LIN {X 0,Y 377.253,Z 474.78,A -85,B 0,C 180,E1 17667.471,E2 17667.471} C_VEL
LIN {X 0,Y 377.352,Z 476.669,A -85,B 0,C 180,E1 17678.06,E2 17678.06} C_VEL
LIN {X 0,Y 405.351,Z 515.448,A -85,B 0,C 180,E1 17684.462,E2 17684.462} C_VEL
LIN {X 0,Y 431.336,Z 545.833,A -85,B 0,C 180,E1 17691.711,E2 17691.711} C_VEL
LIN {X 0,Y 454.819,Z 571.984,A -85,B 0,C 180,E1 17699.556,E2 17699.556} C_VEL
LIN {X 0,Y 473.643,Z 591.464,A -85,B 0,C 180,E1 17707.256,E2 17707.256} C_VEL
LIN {X 0,Y 486.809,Z 605.487,A -85,B 0,C 180,E1 17714.646,E2 17714.646} C_VEL
LIN {X 0,Y 493.723,Z 611.989,A -85,B 0,C 180,E1 17720.274,E2 17720.274} C_VEL
LIN {X 0,Y 498.301,Z 615.614,A -85,B 0,C 180,E1 17727.82,E2 17727.82} C_VEL
LIN {X 0,Y 497.056,Z 614.877,A -85,B 0,C 180,E1 17735.239,E2 17735.239} C_VEL
LIN {X 0,Y 492.043,Z 609.419,A -85,B 0,C 180,E1 17741.556,E2 17741.556} C_VEL
LIN {X 0,Y 481.093,Z 598.897,A -85,B 0,C 180,E1 17748.962,E2 17748.962} C_VEL
LIN {X 0,Y 464.615,Z 582.345,A -85,B 0,C 180,E1 17756.667,E2 17756.667} C_VEL
LIN {X 0,Y 442.794,Z 559.28,A -85,B 0,C 180,E1 17764.614,E2 17764.614} C_VEL
LIN {X 0,Y 416.817,Z 529.891,A -85,B 0,C 180,E1 17772.484,E2 17772.484} C_VEL
LIN {X 0,Y 391.726,Z 498.659,A -85,B 0,C 180,E1 17778.671,E2 17778.671} C_VEL
LIN {X 0,Y 376.899,Z 474.78,A -85,B 0,C 180,E1 17782.231,E2 17782.231} C_VEL
LIN {X 0,Y 377.23,Z 474.78,A -85,B 0,C 180,E1 17792.527,E2 17792.527} C_VEL
LIN {X 0,Y 377.899,Z 474.78,A -85,B 0,C 180,E1 17802.548,E2 17802.548} C_VEL
LIN {X 0,Y 378.35,Z 474.78,A -85,B 0,C 180,E1 17812.001,E2 17812.001} C_VEL
LIN {X 0,Y 378.531,Z 474.78,A -85,B 0,C 180,E1 17821.217,E2 17821.217} C_VEL
LIN {X 0,Y 378.086,Z 474.78,A -85,B 0,C 180,E1 17830.677,E2 17830.677} C_VEL
LIN {X 0,Y 377.317,Z 474.78,A -85,B 0,C 180,E1 17842.532,E2 17842.532} C_VEL
LIN {X 0,Y 376.834,Z 474.78,A -85,B 0,C 180,E1 17853.007,E2 17853.007} C_VEL
LIN {X 0,Y 376.964,Z 476.24,A -85,B 0,C 180,E1 17857.663,E2 17857.663} C_VEL
LIN {X 0,Y 410.937,Z 533.681,A -85,B 0,C 180,E1 17865.009,E2 17865.009} C_VEL
LIN {X 0,Y 427.352,Z 580.89,A -85,B 0,C 180,E1 17869.565,E2 17869.565} C_VEL
LIN {X 0,Y 414.888,Z 639.247,A -85,B 0,C 180,E1 17873.387,E2 17873.387} C_VEL
LIN {X 0,Y 400.436,Z 690.553,A -85,B 0,C 180,E1 17879.252,E2 17879.252} C_VEL
LIN {X 0,Y 388.051,Z 731.295,A -85,B 0,C 180,E1 17887.04,E2 17887.04} C_VEL
LIN {X 0,Y 381.14,Z 758.804,A -85,B 0,C 180,E1 17896.188,E2 17896.188} C_VEL
LIN {X 0,Y 379.523,Z 770.88,A -85,B 0,C 180,E1 17904.267,E2 17904.267} C_VEL
LIN {X 0,Y 379.67,Z 772.444,A -85,B 0,C 180,E1 17913.435,E2 17913.435} C_VEL
LIN {X 0,Y 380.683,Z 761.252,A -85,B 0,C 180,E1 17922.656,E2 17922.656} C_VEL
LIN {X 0,Y 386.704,Z 735.531,A -85,B 0,C 180,E1 17931.873,E2 17931.873} C_VEL
LIN {X 0,Y 398.727,Z 695.822,A -85,B 0,C 180,E1 17939.946,E2 17939.946} C_VEL
LIN {X 0,Y 413.364,Z 644.727,A -85,B 0,C 180,E1 17946.115,E2 17946.115} C_VEL
LIN {X 0,Y 426.272,Z 586.242,A -85,B 0,C 180,E1 17950.179,E2 17950.179} C_VEL
LIN {X 0,Y 425.879,Z 572.479,A -85,B 0,C 180,E1 17951.13,E2 17951.13} C_VEL
LIN {X 0,Y 411.196,Z 534.238,A -85,B 0,C 180,E1 17954.932,E2 17954.932} C_VEL
LIN {X 0,Y 393.3,Z 514.558,A -85,B 0,C 180,E1 17958.309,E2 17958.309} C_VEL
LIN {X 0,Y 369.121,Z 474.78,A -85,B 0,C 180,E1 17963.991,E2 17963.991} C_VEL
LIN {X 0,Y 369.27,Z 474.78,A -85,B 0,C 180,E1 17974.365,E2 17974.365} C_VEL
LIN {X 0,Y 369.746,Z 474.78,A -85,B 0,C 180,E1 17984.544,E2 17984.544} C_VEL
LIN {X 0,Y 370.837,Z 474.78,A -85,B 0,C 180,E1 17996.411,E2 17996.411} C_VEL
LIN {X 0,Y 370.594,Z 474.78,A -85,B 0,C 180,E1 18005.804,E2 18005.804} C_VEL
LIN {X 0,Y 369.536,Z 474.78,A -85,B 0,C 180,E1 18017.86,E2 18017.86} C_VEL
LIN {X 0,Y 369.179,Z 474.78,A -85,B 0,C 180,E1 18028.124,E2 18028.124} C_VEL
LIN {X 0,Y 369.275,Z 476.262,A -85,B 0,C 180,E1 18036.407,E2 18036.407} C_VEL
LIN {X 0,Y 401.233,Z 521.524,A -85,B 0,C 180,E1 18043.923,E2 18043.923} C_VEL
LIN {X 0,Y 427.718,Z 552.348,A -85,B 0,C 180,E1 18051.264,E2 18051.264} C_VEL
LIN {X 0,Y 451.496,Z 578.814,A -85,B 0,C 180,E1 18059.185,E2 18059.185} C_VEL
LIN {X 0,Y 470.182,Z 597.857,A -85,B 0,C 180,E1 18066.735,E2 18066.735} C_VEL
LIN {X 0,Y 484.109,Z 612.956,A -85,B 0,C 180,E1 18074.558,E2 18074.558} C_VEL
LIN {X 0,Y 491.06,Z 619.51,A -85,B 0,C 180,E1 18080.221,E2 18080.221} C_VEL
LIN {X 0,Y 495.609,Z 622.979,A -85,B 0,C 180,E1 18087.369,E2 18087.369} C_VEL
LIN {X 0,Y 494.563,Z 622.493,A -85,B 0,C 180,E1 18095.054,E2 18095.054} C_VEL
LIN {X 0,Y 488.649,Z 616.167,A -85,B 0,C 180,E1 18102.28,E2 18102.28} C_VEL
LIN {X 0,Y 477.592,Z 605.888,A -85,B 0,C 180,E1 18109.476,E2 18109.476} C_VEL
LIN {X 0,Y 460.59,Z 588.514,A -85,B 0,C 180,E1 18117.328,E2 18117.328} C_VEL
LIN {X 0,Y 438.778,Z 565.176,A -85,B 0,C 180,E1 18125.211,E2 18125.211} C_VEL
LIN {X 0,Y 412.727,Z 535.843,A -85,B 0,C 180,E1 18133.033,E2 18133.033} C_VEL
LIN {X 0,Y 387.12,Z 503.729,A -85,B 0,C 180,E1 18139.336,E2 18139.336} C_VEL
LIN {X 0,Y 368.91,Z 474.78,A -85,B 0,C 180,E1 18144.099,E2 18144.099} C_VEL
LIN {X 0,Y 369.287,Z 474.78,A -85,B 0,C 180,E1 18154.522,E2 18154.522} C_VEL
LIN {X 0,Y 370.396,Z 474.78,A -85,B 0,C 180,E1 18167.052,E2 18167.052} C_VEL
LIN {X 0,Y 370.787,Z 474.78,A -85,B 0,C 180,E1 18178.898,E2 18178.898} C_VEL
LIN {X 0,Y 370.229,Z 474.78,A -85,B 0,C 180,E1 18188.318,E2 18188.318} C_VEL
LIN {X 0,Y 369.547,Z 474.78,A -85,B 0,C 180,E1 18198.008,E2 18198.008} C_VEL
LIN {X 0,Y 369.034,Z 474.78,A -85,B 0,C 180,E1 18208.296,E2 18208.296} C_VEL
LIN {X 0,Y 369,Z 476.492,A -85,B 0,C 180,E1 18216.048,E2 18216.048} C_VEL
LIN {X 0,Y 402.556,Z 531.828,A -85,B 0,C 180,E1 18223.735,E2 18223.735} C_VEL
LIN {X 0,Y 421.023,Z 582.01,A -85,B 0,C 180,E1 18228.921,E2 18228.921} C_VEL
LIN {X 0,Y 407.865,Z 641.173,A -85,B 0,C 180,E1 18232.902,E2 18232.902} C_VEL
LIN {X 0,Y 392.907,Z 692.253,A -85,B 0,C 180,E1 18238.92,E2 18238.92} C_VEL
LIN {X 0,Y 379.873,Z 733.361,A -85,B 0,C 180,E1 18247.116,E2 18247.116} C_VEL
LIN {X 0,Y 372.996,Z 759.892,A -85,B 0,C 180,E1 18256.48,E2 18256.48} C_VEL
LIN {X 0,Y 371.54,Z 770.704,A -85,B 0,C 180,E1 18264.143,E2 18264.143} C_VEL
LIN {X 0,Y 371.666,Z 772.269,A -85,B 0,C 180,E1 18273.509,E2 18273.509} C_VEL
LIN {X 0,Y 372.745,Z 761.075,A -85,B 0,C 180,E1 18282.93,E2 18282.93} C_VEL
LIN {X 0,Y 379.147,Z 735.353,A -85,B 0,C 180,E1 18292.332,E2 18292.332} C_VEL
LIN {X 0,Y 391.684,Z 695.644,A -85,B 0,C 180,E1 18300.541,E2 18300.541} C_VEL
LIN {X 0,Y 406.699,Z 645.156,A -85,B 0,C 180,E1 18306.728,E2 18306.728} C_VEL
LIN {X 0,Y 420.12,Z 586.399,A -85,B 0,C 180,E1 18310.867,E2 18310.867} C_VEL
LIN {X 0,Y 417.723,Z 569.296,A -85,B 0,C 180,E1 18312.297,E2 18312.297} C_VEL
LIN {X 0,Y 394.772,Z 517.152,A -85,B 0,C 180,E1 18317.987,E2 18317.987} C_VEL
LIN {X 0,Y 393.3,Z 514.558,A -85,B 0,C 180,E1 18318.309,E2 18318.309} C_VEL
LIN {X 0,Y 379.979,Z 504.983,A -85,B 0,C 180,E1 18320.906,E2 18320.906} C_VEL
LIN {X 0,Y 361.179,Z 474.78,A -85,B 0,C 180,E1 18325.946,E2 18325.946} C_VEL
LIN {X 0,Y 361.25,Z 474.78,A -85,B 0,C 180,E1 18336.406,E2 18336.406} C_VEL
LIN {X 0,Y 361.842,Z 474.78,A -85,B 0,C 180,E1 18346.593,E2 18346.593} C_VEL
LIN {X 0,Y 362.837,Z 474.78,A -85,B 0,C 180,E1 18358.73,E2 18358.73} C_VEL
LIN {X 0,Y 362.068,Z 474.78,A -85,B 0,C 180,E1 18370.175,E2 18370.175} C_VEL
LIN {X 0,Y 361.367,Z 474.78,A -85,B 0,C 180,E1 18380.831,E2 18380.831} C_VEL
LIN {X 0,Y 361.09,Z 474.78,A -85,B 0,C 180,E1 18391.598,E2 18391.598} C_VEL
LIN {X 0,Y 361.379,Z 476.69,A -85,B 0,C 180,E1 18394.678,E2 18394.678} C_VEL
LIN {X 0,Y 398.53,Z 529.166,A -85,B 0,C 180,E1 18403.783,E2 18403.783} C_VEL
LIN {X 0,Y 425.221,Z 560.12,A -85,B 0,C 180,E1 18411.235,E2 18411.235} C_VEL
LIN {X 0,Y 447.851,Z 585.572,A -85,B 0,C 180,E1 18418.807,E2 18418.807} C_VEL
LIN {X 0,Y 467.094,Z 605.139,A -85,B 0,C 180,E1 18426.572,E2 18426.572} C_VEL
LIN {X 0,Y 480.632,Z 619.846,A -85,B 0,C 180,E1 18434.123,E2 18434.123} C_VEL
LIN {X 0,Y 488.105,Z 626.919,A -85,B 0,C 180,E1 18440.161,E2 18440.161} C_VEL
LIN {X 0,Y 492.722,Z 630.41,A -85,B 0,C 180,E1 18447.354,E2 18447.354} C_VEL
LIN {X 0,Y 491.965,Z 630.133,A -85,B 0,C 180,E1 18454.42,E2 18454.42} C_VEL
LIN {X 0,Y 486.457,Z 624.369,A -85,B 0,C 180,E1 18461.691,E2 18461.691} C_VEL
LIN {X 0,Y 476.693,Z 614.961,A -85,B 0,C 180,E1 18468.473,E2 18468.473} C_VEL
LIN {X 0,Y 461.294,Z 600.197,A -85,B 0,C 180,E1 18475.879,E2 18475.879} C_VEL
LIN {X 0,Y 440.846,Z 578.023,A -85,B 0,C 180,E1 18483.666,E2 18483.666} C_VEL
LIN {X 0,Y 415.445,Z 549.712,A -85,B 0,C 180,E1 18491.62,E2 18491.62} C_VEL
LIN {X 0,Y 389.627,Z 518.406,A -85,B 0,C 180,E1 18498.359,E2 18498.359} C_VEL
LIN {X 0,Y 360.885,Z 474.78,A -85,B 0,C 180,E1 18505.78,E2 18505.78} C_VEL
LIN {X 0,Y 361.347,Z 474.78,A -85,B 0,C 180,E1 18516.57,E2 18516.57} C_VEL
LIN {X 0,Y 362.325,Z 474.78,A -85,B 0,C 180,E1 18526.759,E2 18526.759} C_VEL
LIN {X 0,Y 362.785,Z 474.78,A -85,B 0,C 180,E1 18538.874,E2 18538.874} C_VEL
LIN {X 0,Y 362.088,Z 474.78,A -85,B 0,C 180,E1 18550.192,E2 18550.192} C_VEL
LIN {X 0,Y 361.315,Z 474.78,A -85,B 0,C 180,E1 18560.989,E2 18560.989} C_VEL
LIN {X 0,Y 360.794,Z 474.78,A -85,B 0,C 180,E1 18571.797,E2 18571.797} C_VEL
LIN {X 0,Y 360.916,Z 476.34,A -85,B 0,C 180,E1 18574.251,E2 18574.251} C_VEL
LIN {X 0,Y 393.845,Z 529.31,A -85,B 0,C 180,E1 18582.291,E2 18582.291} C_VEL
LIN {X 0,Y 414.012,Z 581.264,A -85,B 0,C 180,E1 18588.03,E2 18588.03} C_VEL
LIN {X 0,Y 401.712,Z 640.094,A -85,B 0,C 180,E1 18592.121,E2 18592.121} C_VEL
LIN {X 0,Y 385.949,Z 692.075,A -85,B 0,C 180,E1 18598.296,E2 18598.296} C_VEL
LIN {X 0,Y 372.408,Z 733.144,A -85,B 0,C 180,E1 18606.619,E2 18606.619} C_VEL
LIN {X 0,Y 365.12,Z 759.714,A -85,B 0,C 180,E1 18616.183,E2 18616.183} C_VEL
LIN {X 0,Y 363.54,Z 770.529,A -85,B 0,C 180,E1 18624.014,E2 18624.014} C_VEL
LIN {X 0,Y 363.652,Z 772.094,A -85,B 0,C 180,E1 18633.586,E2 18633.586} C_VEL
LIN {X 0,Y 364.827,Z 760.897,A -85,B 0,C 180,E1 18643.216,E2 18643.216} C_VEL
LIN {X 0,Y 371.615,Z 735.174,A -85,B 0,C 180,E1 18652.81,E2 18652.81} C_VEL
LIN {X 0,Y 384.684,Z 695.466,A -85,B 0,C 180,E1 18661.158,E2 18661.158} C_VEL
LIN {X 0,Y 400.187,Z 645.172,A -85,B 0,C 180,E1 18667.402,E2 18667.402} C_VEL
LIN {X 0,Y 414.019,Z 586.453,A -85,B 0,C 180,E1 18671.585,E2 18671.585} C_VEL
LIN {X 0,Y 401.458,Z 545.316,A -85,B 0,C 180,E1 18675.833,E2 18675.833} C_VEL
LIN {X 0,Y 379.979,Z 504.983,A -85,B 0,C 180,E1 18680.906,E2 18680.906} C_VEL
LIN {X 0,Y 366.931,Z 496.837,A -85,B 0,C 180,E1 18683.733,E2 18683.733} C_VEL
LIN {X 0,Y 353.212,Z 474.78,A -85,B 0,C 180,E1 18688.033,E2 18688.033} C_VEL
LIN {X 0,Y 353.277,Z 474.78,A -85,B 0,C 180,E1 18698.51,E2 18698.51} C_VEL
LIN {X 0,Y 354.024,Z 474.78,A -85,B 0,C 180,E1 18708.806,E2 18708.806} C_VEL
LIN {X 0,Y 354.837,Z 474.78,A -85,B 0,C 180,E1 18718.702,E2 18718.702} C_VEL
LIN {X 0,Y 354.17,Z 474.78,A -85,B 0,C 180,E1 18728.549,E2 18728.549} C_VEL
LIN {X 0,Y 353.411,Z 474.78,A -85,B 0,C 180,E1 18738.705,E2 18738.705} C_VEL
LIN {X 0,Y 353.081,Z 474.78,A -85,B 0,C 180,E1 18749.53,E2 18749.53} C_VEL
LIN {X 0,Y 353.185,Z 476.506,A -85,B 0,C 180,E1 18752.688,E2 18752.688} C_VEL
LIN {X 0,Y 395.397,Z 536.478,A -85,B 0,C 180,E1 18763.601,E2 18763.601} C_VEL
LIN {X 0,Y 421.763,Z 567.154,A -85,B 0,C 180,E1 18771.007,E2 18771.007} C_VEL
LIN {X 0,Y 444.377,Z 592.548,A -85,B 0,C 180,E1 18778.57,E2 18778.57} C_VEL
LIN {X 0,Y 463.314,Z 611.985,A -85,B 0,C 180,E1 18786.219,E2 18786.219} C_VEL
LIN {X 0,Y 476.243,Z 626.049,A -85,B 0,C 180,E1 18793.347,E2 18793.347} C_VEL
LIN {X 0,Y 484.87,Z 634.18,A -85,B 0,C 180,E1 18800.095,E2 18800.095} C_VEL
LIN {X 0,Y 489.538,Z 637.751,A -85,B 0,C 180,E1 18807.337,E2 18807.337} C_VEL
LIN {X 0,Y 488.768,Z 637.437,A -85,B 0,C 180,E1 18814.449,E2 18814.449} C_VEL
LIN {X 0,Y 483.23,Z 631.64,A -85,B 0,C 180,E1 18821.77,E2 18821.77} C_VEL
LIN {X 0,Y 472.737,Z 621.628,A -85,B 0,C 180,E1 18828.947,E2 18828.947} C_VEL
LIN {X 0,Y 456.557,Z 605.758,A -85,B 0,C 180,E1 18836.642,E2 18836.642} C_VEL
LIN {X 0,Y 435.27,Z 582.988,A -85,B 0,C 180,E1 18844.583,E2 18844.583} C_VEL
LIN {X 0,Y 409.701,Z 553.731,A -85,B 0,C 180,E1 18852.534,E2 18852.534} C_VEL
LIN {X 0,Y 384.049,Z 522.559,A -85,B 0,C 180,E1 18859.129,E2 18859.129} C_VEL
LIN {X 0,Y 352.898,Z 474.78,A -85,B 0,C 180,E1 18867.58,E2 18867.58} C_VEL
LIN {X 0,Y 353.441,Z 474.78,A -85,B 0,C 180,E1 18878.679,E2 18878.679} C_VEL
LIN {X 0,Y 354.377,Z 474.78,A -85,B 0,C 180,E1 18888.967,E2 18888.967} C_VEL
LIN {X 0,Y 354.792,Z 474.78,A -85,B 0,C 180,E1 18898.848,E2 18898.848} C_VEL
LIN {X 0,Y 354.173,Z 474.78,A -85,B 0,C 180,E1 18908.697,E2 18908.697} C_VEL
LIN {X 0,Y 353.419,Z 474.78,A -85,B 0,C 180,E1 18918.86,E2 18918.86} C_VEL
LIN {X 0,Y 352.786,Z 474.78,A -85,B 0,C 180,E1 18931.278,E2 18931.278} C_VEL
LIN {X 0,Y 353.154,Z 477.279,A -85,B 0,C 180,E1 18932.402,E2 18932.402} C_VEL
LIN {X 0,Y 383.773,Z 524.559,A -85,B 0,C 180,E1 18940.433,E2 18940.433} C_VEL
LIN {X 0,Y 404.628,Z 573.54,A -85,B 0,C 180,E1 18946.297,E2 18946.297} C_VEL
LIN {X 0,Y 407.449,Z 590.108,A -85,B 0,C 180,E1 18947.882,E2 18947.882} C_VEL
LIN {X 0,Y 392.946,Z 647.964,A -85,B 0,C 180,E1 18952.172,E2 18952.172} C_VEL
LIN {X 0,Y 377.233,Z 696.977,A -85,B 0,C 180,E1 18958.493,E2 18958.493} C_VEL
LIN {X 0,Y 363.844,Z 736.024,A -85,B 0,C 180,E1 18966.999,E2 18966.999} C_VEL
LIN {X 0,Y 356.987,Z 760.721,A -85,B 0,C 180,E1 18976.488,E2 18976.488} C_VEL
LIN {X 0,Y 355.331,Z 771.911,A -85,B 0,C 180,E1 18986.329,E2 18986.329} C_VEL
LIN {X 0,Y 355.638,Z 771.918,A -85,B 0,C 180,E1 18993.667,E2 18993.667} C_VEL
LIN {X 0,Y 356.922,Z 760.719,A -85,B 0,C 180,E1 19003.514,E2 19003.514} C_VEL
LIN {X 0,Y 364.133,Z 734.997,A -85,B 0,C 180,E1 19013.306,E2 19013.306} C_VEL
LIN {X 0,Y 377.765,Z 695.289,A -85,B 0,C 180,E1 19021.795,E2 19021.795} C_VEL
LIN {X 0,Y 393.994,Z 644.281,A -85,B 0,C 180,E1 19028.187,E2 19028.187} C_VEL
LIN {X 0,Y 407.973,Z 585.436,A -85,B 0,C 180,E1 19032.406,E2 19032.406} C_VEL
LIN {X 0,Y 389.397,Z 535.247,A -85,B 0,C 180,E1 19038.149,E2 19038.149} C_VEL
LIN {X 0,Y 366.931,Z 496.837,A -85,B 0,C 180,E1 19043.733,E2 19043.733} C_VEL
LIN {X 0,Y 354.564,Z 489.645,A -85,B 0,C 180,E1 19046.794,E2 19046.794} C_VEL
LIN {X 0,Y 345.176,Z 474.78,A -85,B 0,C 180,E1 19050.264,E2 19050.264} C_VEL
LIN {X 0,Y 345.393,Z 474.78,A -85,B 0,C 180,E1 19060.731,E2 19060.731} C_VEL
LIN {X 0,Y 346.103,Z 474.78,A -85,B 0,C 180,E1 19071.098,E2 19071.098} C_VEL
LIN {X 0,Y 346.577,Z 474.78,A -85,B 0,C 180,E1 19081.179,E2 19081.179} C_VEL
LIN {X 0,Y 345.967,Z 474.78,A -85,B 0,C 180,E1 19091.305,E2 19091.305} C_VEL
LIN {X 0,Y 345.246,Z 474.78,A -85,B 0,C 180,E1 19101.853,E2 19101.853} C_VEL
LIN {X 0,Y 345.226,Z 476.748,A -85,B 0,C 180,E1 19110.565,E2 19110.565} C_VEL
LIN {X 0,Y 380.994,Z 530.05,A -85,B 0,C 180,E1 19120.704,E2 19120.704} C_VEL
LIN {X 0,Y 407.52,Z 561.948,A -85,B 0,C 180,E1 19127.633,E2 19127.633} C_VEL
LIN {X 0,Y 432.358,Z 590.354,A -85,B 0,C 180,E1 19135.447,E2 19135.447} C_VEL
LIN {X 0,Y 452.771,Z 612.44,A -85,B 0,C 180,E1 19143.118,E2 19143.118} C_VEL
LIN {X 0,Y 469.075,Z 628.804,A -85,B 0,C 180,E1 19150.916,E2 19150.916} C_VEL
LIN {X 0,Y 479.779,Z 638.684,A -85,B 0,C 180,E1 19158.144,E2 19158.144} C_VEL
LIN {X 0,Y 485.235,Z 644.657,A -85,B 0,C 180,E1 19165.519,E2 19165.519} C_VEL
LIN {X 0,Y 485.863,Z 645.146,A -85,B 0,C 180,E1 19172.684,E2 19172.684} C_VEL
LIN {X 0,Y 481.306,Z 641.368,A -85,B 0,C 180,E1 19179.979,E2 19179.979} C_VEL
LIN {X 0,Y 472.784,Z 633.007,A -85,B 0,C 180,E1 19186.761,E2 19186.761} C_VEL
LIN {X 0,Y 458.197,Z 617.953,A -85,B 0,C 180,E1 19194.549,E2 19194.549} C_VEL
LIN {X 0,Y 438.324,Z 597.323,A -85,B 0,C 180,E1 19202.429,E2 19202.429} C_VEL
LIN {X 0,Y 413.532,Z 569.562,A -85,B 0,C 180,E1 19210.544,E2 19210.544} C_VEL
LIN {X 0,Y 386.706,Z 537.744,A -85,B 0,C 180,E1 19217.882,E2 19217.882} C_VEL
LIN {X 0,Y 346.919,Z 480.176,A -85,B 0,C 180,E1 19228.827,E2 19228.827} C_VEL
LIN {X 0,Y 344.875,Z 474.78,A -85,B 0,C 180,E1 19229.695,E2 19229.695} C_VEL
LIN {X 0,Y 345.585,Z 474.78,A -85,B 0,C 180,E1 19240.855,E2 19240.855} C_VEL
LIN {X 0,Y 346.296,Z 474.78,A -85,B 0,C 180,E1 19251.255,E2 19251.255} C_VEL
LIN {X 0,Y 346.545,Z 474.78,A -85,B 0,C 180,E1 19261.329,E2 19261.329} C_VEL
LIN {X 0,Y 345.961,Z 474.78,A -85,B 0,C 180,E1 19271.459,E2 19271.459} C_VEL
LIN {X 0,Y 345.161,Z 474.78,A -85,B 0,C 180,E1 19282.021,E2 19282.021} C_VEL
LIN {X 0,Y 344.998,Z 476.44,A -85,B 0,C 180,E1 19290.18,E2 19290.18} C_VEL
LIN {X 0,Y 375.949,Z 523.84,A -85,B 0,C 180,E1 19298.996,E2 19298.996} C_VEL
LIN {X 0,Y 396.866,Z 571.664,A -85,B 0,C 180,E1 19305.105,E2 19305.105} C_VEL
LIN {X 0,Y 400.882,Z 593.099,A -85,B 0,C 180,E1 19307.276,E2 19307.276} C_VEL
LIN {X 0,Y 385.572,Z 651.329,A -85,B 0,C 180,E1 19311.789,E2 19311.789} C_VEL
LIN {X 0,Y 369.071,Z 700.172,A -85,B 0,C 180,E1 19318.406,E2 19318.406} C_VEL
LIN {X 0,Y 355.79,Z 737.432,A -85,B 0,C 180,E1 19326.961,E2 19326.961} C_VEL
LIN {X 0,Y 348.864,Z 761.569,A -85,B 0,C 180,E1 19336.808,E2 19336.808} C_VEL
LIN {X 0,Y 347.329,Z 771.736,A -85,B 0,C 180,E1 19346.245,E2 19346.245} C_VEL
LIN {X 0,Y 347.624,Z 771.743,A -85,B 0,C 180,E1 19353.752,E2 19353.752} C_VEL
LIN {X 0,Y 349.033,Z 760.542,A -85,B 0,C 180,E1 19363.825,E2 19363.825} C_VEL
LIN {X 0,Y 356.659,Z 734.819,A -85,B 0,C 180,E1 19373.824,E2 19373.824} C_VEL
LIN {X 0,Y 370.853,Z 695.11,A -85,B 0,C 180,E1 19382.459,E2 19382.459} C_VEL
LIN {X 0,Y 387.687,Z 644.096,A -85,B 0,C 180,E1 19388.925,E2 19388.925} C_VEL
LIN {X 0,Y 401.082,Z 586.026,A -85,B 0,C 180,E1 19393.25,E2 19393.25} C_VEL
LIN {X 0,Y 382.37,Z 535.929,A -85,B 0,C 180,E1 19399.294,E2 19399.294} C_VEL
LIN {X 0,Y 354.564,Z 489.645,A -85,B 0,C 180,E1 19406.794,E2 19406.794} C_VEL
LIN {X 0,Y 342.781,Z 484.519,A -85,B 0,C 180,E1 19410.126,E2 19410.126} C_VEL
LIN {X 0,Y 337.096,Z 474.78,A -85,B 0,C 180,E1 19412.669,E2 19412.669} C_VEL
LIN {X 0,Y 337.66,Z 474.78,A -85,B 0,C 180,E1 19425.613,E2 19425.613} C_VEL
LIN {X 0,Y 338.76,Z 474.78,A -85,B 0,C 180,E1 19436.071,E2 19436.071} C_VEL
LIN {X 0,Y 338.452,Z 474.78,A -85,B 0,C 180,E1 19446.357,E2 19446.357} C_VEL
LIN {X 0,Y 337.479,Z 474.78,A -85,B 0,C 180,E1 19456.91,E2 19456.91} C_VEL
LIN {X 0,Y 337.116,Z 476.425,A -85,B 0,C 180,E1 19468.113,E2 19468.113} C_VEL
LIN {X 0,Y 364.232,Z 516.802,A -85,B 0,C 180,E1 19476.787,E2 19476.787} C_VEL
LIN {X 0,Y 394.343,Z 558.16,A -85,B 0,C 180,E1 19484.857,E2 19484.857} C_VEL
LIN {X 0,Y 419.895,Z 587.512,A -85,B 0,C 180,E1 19492.396,E2 19492.396} C_VEL
LIN {X 0,Y 441.859,Z 611.989,A -85,B 0,C 180,E1 19500.156,E2 19500.156} C_VEL
LIN {X 0,Y 459.243,Z 630.088,A -85,B 0,C 180,E1 19507.682,E2 19507.682} C_VEL
LIN {X 0,Y 471.928,Z 642.653,A -85,B 0,C 180,E1 19515.104,E2 19515.104} C_VEL
LIN {X 0,Y 478.998,Z 650.073,A -85,B 0,C 180,E1 19521.809,E2 19521.809} C_VEL
LIN {X 0,Y 482.498,Z 652.472,A -85,B 0,C 180,E1 19529.1,E2 19529.1} C_VEL
LIN {X 0,Y 480.464,Z 650.929,A -85,B 0,C 180,E1 19536.402,E2 19536.402} C_VEL
LIN {X 0,Y 473.453,Z 643.633,A -85,B 0,C 180,E1 19543.9,E2 19543.9} C_VEL
LIN {X 0,Y 460.324,Z 631.457,A -85,B 0,C 180,E1 19551.722,E2 19551.722} C_VEL
LIN {X 0,Y 443.156,Z 613.602,A -85,B 0,C 180,E1 19559.307,E2 19559.307} C_VEL
LIN {X 0,Y 420.917,Z 589.125,A -85,B 0,C 180,E1 19567.215,E2 19567.215} C_VEL
LIN {X 0,Y 395.255,Z 559.867,A -85,B 0,C 180,E1 19574.848,E2 19574.848} C_VEL
LIN {X 0,Y 363.971,Z 516.669,A -85,B 0,C 180,E1 19583.275,E2 19583.275} C_VEL
LIN {X 0,Y 339.185,Z 480.396,A -85,B 0,C 180,E1 19591.064,E2 19591.064} C_VEL
LIN {X 0,Y 336.995,Z 474.78,A -85,B 0,C 180,E1 19592.314,E2 19592.314} C_VEL
LIN {X 0,Y 337.965,Z 474.78,A -85,B 0,C 180,E1 19604.738,E2 19604.738} C_VEL
LIN {X 0,Y 338.735,Z 474.78,A -85,B 0,C 180,E1 19616.733,E2 19616.733} C_VEL
LIN {X 0,Y 338.404,Z 474.78,A -85,B 0,C 180,E1 19626.513,E2 19626.513} C_VEL
LIN {X 0,Y 337.47,Z 474.78,A -85,B 0,C 180,E1 19637.072,E2 19637.072} C_VEL
LIN {X 0,Y 337.086,Z 476.411,A -85,B 0,C 180,E1 19647.795,E2 19647.795} C_VEL
LIN {X 0,Y 366.168,Z 519.911,A -85,B 0,C 180,E1 19656.924,E2 19656.924} C_VEL
LIN {X 0,Y 388.11,Z 566.586,A -85,B 0,C 180,E1 19663.458,E2 19663.458} C_VEL
LIN {X 0,Y 394.595,Z 594.757,A -85,B 0,C 180,E1 19666.591,E2 19666.591} C_VEL
LIN {X 0,Y 378.986,Z 652.005,A -85,B 0,C 180,E1 19671.117,E2 19671.117} C_VEL
LIN {X 0,Y 361.501,Z 701.793,A -85,B 0,C 180,E1 19678.044,E2 19678.044} C_VEL
LIN {X 0,Y 347.511,Z 739.493,A -85,B 0,C 180,E1 19687.121,E2 19687.121} C_VEL
LIN {X 0,Y 340.765,Z 762.418,A -85,B 0,C 180,E1 19697.143,E2 19697.143} C_VEL
LIN {X 0,Y 339.357,Z 771.561,A -85,B 0,C 180,E1 19706.156,E2 19706.156} C_VEL
LIN {X 0,Y 339.617,Z 771.567,A -85,B 0,C 180,E1 19713.84,E2 19713.84} C_VEL
LIN {X 0,Y 341.169,Z 760.365,A -85,B 0,C 180,E1 19724.151,E2 19724.151} C_VEL
LIN {X 0,Y 349.217,Z 734.64,A -85,B 0,C 180,E1 19734.364,E2 19734.364} C_VEL
LIN {X 0,Y 363.734,Z 695.662,A -85,B 0,C 180,E1 19743.021,E2 19743.021} C_VEL
LIN {X 0,Y 381.011,Z 645.267,A -85,B 0,C 180,E1 19749.555,E2 19749.555} C_VEL
LIN {X 0,Y 394.563,Z 588.059,A -85,B 0,C 180,E1 19753.967,E2 19753.967} C_VEL
LIN {X 0,Y 376.403,Z 538.545,A -85,B 0,C 180,E1 19760.22,E2 19760.22} C_VEL
LIN {X 0,Y 349.381,Z 493.73,A -85,B 0,C 180,E1 19767.954,E2 19767.954} C_VEL
LIN {X 0,Y 342.781,Z 484.519,A -85,B 0,C 180,E1 19770.126,E2 19770.126} C_VEL
LIN {X 0,Y 331.939,Z 480.931,A -85,B 0,C 180,E1 19773.712,E2 19773.712} C_VEL
LIN {X 0,Y 329.046,Z 474.78,A -85,B 0,C 180,E1 19775.395,E2 19775.395} C_VEL
LIN {X 0,Y 329.852,Z 474.78,A -85,B 0,C 180,E1 19787.974,E2 19787.974} C_VEL
LIN {X 0,Y 330.827,Z 474.78,A -85,B 0,C 180,E1 19798.607,E2 19798.607} C_VEL
LIN {X 0,Y 330.058,Z 474.78,A -85,B 0,C 180,E1 19809.179,E2 19809.179} C_VEL
LIN {X 0,Y 329.216,Z 474.78,A -85,B 0,C 180,E1 19820.137,E2 19820.137} C_VEL
LIN {X 0,Y 329.254,Z 476.439,A -85,B 0,C 180,E1 19825.416,E2 19825.416} C_VEL
LIN {X 0,Y 356.148,Z 515.569,A -85,B 0,C 180,E1 19834.925,E2 19834.925} C_VEL
LIN {X 0,Y 387.954,Z 562.453,A -85,B 0,C 180,E1 19844.053,E2 19844.053} C_VEL
LIN {X 0,Y 414.509,Z 592.723,A -85,B 0,C 180,E1 19851.8,E2 19851.8} C_VEL
LIN {X 0,Y 437.238,Z 618.113,A -85,B 0,C 180,E1 19859.807,E2 19859.807} C_VEL
LIN {X 0,Y 454.937,Z 636.614,A -85,B 0,C 180,E1 19867.459,E2 19867.459} C_VEL
LIN {X 0,Y 467.871,Z 649.503,A -85,B 0,C 180,E1 19875.036,E2 19875.036} C_VEL
LIN {X 0,Y 474.984,Z 656.952,A -85,B 0,C 180,E1 19881.74,E2 19881.74} C_VEL
LIN {X 0,Y 478.465,Z 659.377,A -85,B 0,C 180,E1 19889.092,E2 19889.092} C_VEL
LIN {X 0,Y 476.484,Z 657.859,A -85,B 0,C 180,E1 19896.396,E2 19896.396} C_VEL
LIN {X 0,Y 469.328,Z 650.439,A -85,B 0,C 180,E1 19904.025,E2 19904.025} C_VEL
LIN {X 0,Y 456.816,Z 638.806,A -85,B 0,C 180,E1 19911.552,E2 19911.552} C_VEL
LIN {X 0,Y 439.411,Z 620.702,A -85,B 0,C 180,E1 19919.319,E2 19919.319} C_VEL
LIN {X 0,Y 417.38,Z 596.414,A -85,B 0,C 180,E1 19927.214,E2 19927.214} C_VEL
LIN {X 0,Y 391.558,Z 567.138,A -85,B 0,C 180,E1 19934.94,E2 19934.94} C_VEL
LIN {X 0,Y 359.294,Z 521.478,A -85,B 0,C 180,E1 19944.036,E2 19944.036} C_VEL
LIN {X 0,Y 333.055,Z 481.731,A -85,B 0,C 180,E1 19952.984,E2 19952.984} C_VEL
LIN {X 0,Y 329.121,Z 474.78,A -85,B 0,C 180,E1 19954.847,E2 19954.847} C_VEL
LIN {X 0,Y 330.062,Z 474.78,A -85,B 0,C 180,E1 19965.437,E2 19965.437} C_VEL
LIN {X 0,Y 330.701,Z 474.78,A -85,B 0,C 180,E1 19976.719,E2 19976.719} C_VEL
LIN {X 0,Y 330.36,Z 474.78,A -85,B 0,C 180,E1 19986.672,E2 19986.672} C_VEL
LIN {X 0,Y 329.226,Z 474.78,A -85,B 0,C 180,E1 19999.217,E2 19999.217} C_VEL
LIN {X 0,Y 329.108,Z 476.457,A -85,B 0,C 180,E1 20005.055,E2 20005.055} C_VEL
LIN {X 0,Y 356.122,Z 515.639,A -85,B 0,C 180,E1 20014.549,E2 20014.549} C_VEL
LIN {X 0,Y 379.593,Z 562.455,A -85,B 0,C 180,E1 20021.793,E2 20021.793} C_VEL
LIN {X 0,Y 388.424,Z 596.117,A -85,B 0,C 180,E1 20025.872,E2 20025.872} C_VEL
LIN {X 0,Y 372.303,Z 653.133,A -85,B 0,C 180,E1 20030.472,E2 20030.472} C_VEL
LIN {X 0,Y 354.521,Z 701.942,A -85,B 0,C 180,E1 20037.408,E2 20037.408} C_VEL
LIN {X 0,Y 340.241,Z 738.724,A -85,B 0,C 180,E1 20046.403,E2 20046.403} C_VEL
LIN {X 0,Y 332.851,Z 762.241,A -85,B 0,C 180,E1 20056.832,E2 20056.832} C_VEL
LIN {X 0,Y 331.354,Z 771.386,A -85,B 0,C 180,E1 20066.063,E2 20066.063} C_VEL
LIN {X 0,Y 331.603,Z 771.392,A -85,B 0,C 180,E1 20073.933,E2 20073.933} C_VEL
LIN {X 0,Y 333.316,Z 760.188,A -85,B 0,C 180,E1 20084.491,E2 20084.491} C_VEL
LIN {X 0,Y 342.26,Z 733.436,A -85,B 0,C 180,E1 20095.243,E2 20095.243} C_VEL
LIN {X 0,Y 357.731,Z 693.518,A -85,B 0,C 180,E1 20104.075,E2 20104.075} C_VEL
LIN {X 0,Y 375.694,Z 642.395,A -85,B 0,C 180,E1 20110.608,E2 20110.608} C_VEL
LIN {X 0,Y 388.199,Z 590.482,A -85,B 0,C 180,E1 20114.663,E2 20114.663} C_VEL
LIN {X 0,Y 370.494,Z 541.416,A -85,B 0,C 180,E1 20121.17,E2 20121.17} C_VEL
LIN {X 0,Y 343.502,Z 495.682,A -85,B 0,C 180,E1 20129.468,E2 20129.468} C_VEL
LIN {X 0,Y 331.939,Z 480.931,A -85,B 0,C 180,E1 20133.712,E2 20133.712} C_VEL
LIN {X 0,Y 322.232,Z 478.913,A -85,B 0,C 180,E1 20137.542,E2 20137.542} C_VEL
LIN {X 0,Y 321.119,Z 474.78,A -85,B 0,C 180,E1 20138.673,E2 20138.673} C_VEL
LIN {X 0,Y 322.001,Z 474.78,A -85,B 0,C 180,E1 20150.426,E2 20150.426} C_VEL
LIN {X 0,Y 322.58,Z 474.78,A -85,B 0,C 180,E1 20161.267,E2 20161.267} C_VEL
LIN {X 0,Y 321.815,Z 474.78,A -85,B 0,C 180,E1 20172.166,E2 20172.166} C_VEL
LIN {X 0,Y 321.332,Z 476.753,A -85,B 0,C 180,E1 20182.251,E2 20182.251} C_VEL
LIN {X 0,Y 345.195,Z 509.762,A -85,B 0,C 180,E1 20191.928,E2 20191.928} C_VEL
LIN {X 0,Y 380.421,Z 565.155,A -85,B 0,C 180,E1 20202.984,E2 20202.984} C_VEL
LIN {X 0,Y 407.281,Z 595.802,A -85,B 0,C 180,E1 20210.696,E2 20210.696} C_VEL
LIN {X 0,Y 430.616,Z 621.879,A -85,B 0,C 180,E1 20218.732,E2 20218.732} C_VEL
LIN {X 0,Y 448.98,Z 641.285,A -85,B 0,C 180,E1 20226.507,E2 20226.507} C_VEL
LIN {X 0,Y 461.705,Z 654.853,A -85,B 0,C 180,E1 20233.788,E2 20233.788} C_VEL
LIN {X 0,Y 469.357,Z 662.144,A -85,B 0,C 180,E1 20240.049,E2 20240.049} C_VEL
LIN {X 0,Y 474.009,Z 665.64,A -85,B 0,C 180,E1 20247.249,E2 20247.249} C_VEL
LIN {X 0,Y 473.128,Z 665.29,A -85,B 0,C 180,E1 20254.596,E2 20254.596} C_VEL
LIN {X 0,Y 467.48,Z 659.317,A -85,B 0,C 180,E1 20262.173,E2 20262.173} C_VEL
LIN {X 0,Y 455.723,Z 648.259,A -85,B 0,C 180,E1 20269.996,E2 20269.996} C_VEL
LIN {X 0,Y 439.27,Z 631.503,A -85,B 0,C 180,E1 20277.779,E2 20277.779} C_VEL
LIN {X 0,Y 417.606,Z 608.339,A -85,B 0,C 180,E1 20285.827,E2 20285.827} C_VEL
LIN {X 0,Y 391.843,Z 578.907,A -85,B 0,C 180,E1 20293.846,E2 20293.846} C_VEL
LIN {X 0,Y 358.976,Z 534.282,A -85,B 0,C 180,E1 20303.341,E2 20303.341} C_VEL
LIN {X 0,Y 334.881,Z 495.278,A -85,B 0,C 180,E1 20311.763,E2 20311.763} C_VEL
LIN {X 0,Y 321.264,Z 474.78,A -85,B 0,C 180,E1 20318.618,E2 20318.618} C_VEL
LIN {X 0,Y 322.295,Z 474.78,A -85,B 0,C 180,E1 20330.598,E2 20330.598} C_VEL
LIN {X 0,Y 322.535,Z 474.78,A -85,B 0,C 180,E1 20341.428,E2 20341.428} C_VEL
LIN {X 0,Y 321.789,Z 474.78,A -85,B 0,C 180,E1 20352.332,E2 20352.332} C_VEL
LIN {X 0,Y 321.237,Z 476.711,A -85,B 0,C 180,E1 20361.9,E2 20361.9} C_VEL
LIN {X 0,Y 344.534,Z 508.894,A -85,B 0,C 180,E1 20371.341,E2 20371.341} C_VEL
LIN {X 0,Y 369.302,Z 554.574,A -85,B 0,C 180,E1 20379.45,E2 20379.45} C_VEL
LIN {X 0,Y 382.181,Z 597.948,A -85,B 0,C 180,E1 20385.157,E2 20385.157} C_VEL
LIN {X 0,Y 365.651,Z 654.158,A -85,B 0,C 180,E1 20389.802,E2 20389.802} C_VEL
LIN {X 0,Y 347.19,Z 702.971,A -85,B 0,C 180,E1 20396.908,E2 20396.908} C_VEL
LIN {X 0,Y 332.176,Z 740.166,A -85,B 0,C 180,E1 20406.358,E2 20406.358} C_VEL
LIN {X 0,Y 324.768,Z 763.09,A -85,B 0,C 180,E1 20417.185,E2 20417.185} C_VEL
LIN {X 0,Y 323.351,Z 771.211,A -85,B 0,C 180,E1 20425.966,E2 20425.966} C_VEL
LIN {X 0,Y 323.589,Z 771.216,A -85,B 0,C 180,E1 20434.031,E2 20434.031} C_VEL
LIN {X 0,Y 325.47,Z 760.01,A -85,B 0,C 180,E1 20444.848,E2 20444.848} C_VEL
LIN {X 0,Y 334.902,Z 733.258,A -85,B 0,C 180,E1 20455.838,E2 20455.838} C_VEL
LIN {X 0,Y 351.02,Z 693.341,A -85,B 0,C 180,E1 20464.819,E2 20464.819} C_VEL
LIN {X 0,Y 369.577,Z 642.218,A -85,B 0,C 180,E1 20471.426,E2 20471.426} C_VEL
LIN {X 0,Y 381.966,Z 593.136,A -85,B 0,C 180,E1 20475.349,E2 20475.349} C_VEL
LIN {X 0,Y 364.608,Z 544.031,A -85,B 0,C 180,E1 20482.172,E2 20482.172} C_VEL
LIN {X 0,Y 339.888,Z 501.791,A -85,B 0,C 180,E1 20490.256,E2 20490.256} C_VEL
LIN {X 0,Y 322.232,Z 478.913,A -85,B 0,C 180,E1 20497.542,E2 20497.542} C_VEL
LIN {X 0,Y 313.369,Z 474.78,A -85,B 0,C 180,E1 20503.533,E2 20503.533} C_VEL
LIN {X 0,Y 314.64,Z 474.78,A -85,B 0,C 180,E1 20515.769,E2 20515.769} C_VEL
LIN {X 0,Y 314.31,Z 474.78,A -85,B 0,C 180,E1 20526.848,E2 20526.848} C_VEL
LIN {X 0,Y 313.439,Z 476.456,A -85,B 0,C 180,E1 20538.35,E2 20538.35} C_VEL
LIN {X 0,Y 333.799,Z 504.088,A -85,B 0,C 180,E1 20548.306,E2 20548.306} C_VEL
LIN {X 0,Y 357.919,Z 545.566,A -85,B 0,C 180,E1 20557.228,E2 20557.228} C_VEL
LIN {X 0,Y 390.423,Z 588.434,A -85,B 0,C 180,E1 20566.827,E2 20566.827} C_VEL
LIN {X 0,Y 414.855,Z 616.343,A -85,B 0,C 180,E1 20574.609,E2 20574.609} C_VEL
LIN {X 0,Y 435.636,Z 638.983,A -85,B 0,C 180,E1 20582.506,E2 20582.506} C_VEL
LIN {X 0,Y 451.246,Z 654.849,A -85,B 0,C 180,E1 20589.967,E2 20589.967} C_VEL
LIN {X 0,Y 462.879,Z 665.655,A -85,B 0,C 180,E1 20597.705,E2 20597.705} C_VEL
LIN {X 0,Y 468.58,Z 671.948,A -85,B 0,C 180,E1 20605.359,E2 20605.359} C_VEL
LIN {X 0,Y 469.28,Z 672.453,A -85,B 0,C 180,E1 20612.778,E2 20612.778} C_VEL
LIN {X 0,Y 464.419,Z 668.311,A -85,B 0,C 180,E1 20620.346,E2 20620.346} C_VEL
LIN {X 0,Y 456.19,Z 660.207,A -85,B 0,C 180,E1 20626.969,E2 20626.969} C_VEL
LIN {X 0,Y 442.022,Z 645.475,A -85,B 0,C 180,E1 20634.692,E2 20634.692} C_VEL
LIN {X 0,Y 422.565,Z 625.269,A -85,B 0,C 180,E1 20642.575,E2 20642.575} C_VEL
LIN {X 0,Y 398.827,Z 598.777,A -85,B 0,C 180,E1 20650.562,E2 20650.562} C_VEL
LIN {X 0,Y 370.261,Z 564.69,A -85,B 0,C 180,E1 20658.797,E2 20658.797} C_VEL
LIN {X 0,Y 335.857,Z 507.65,A -85,B 0,C 180,E1 20670.85,E2 20670.85} C_VEL
LIN {X 0,Y 317.053,Z 481.544,A -85,B 0,C 180,E1 20679.431,E2 20679.431} C_VEL
LIN {X 0,Y 313.553,Z 474.78,A -85,B 0,C 180,E1 20681.756,E2 20681.756} C_VEL
LIN {X 0,Y 314.3,Z 474.78,A -85,B 0,C 180,E1 20693.152,E2 20693.152} C_VEL
LIN {X 0,Y 314.564,Z 474.78,A -85,B 0,C 180,E1 20704.232,E2 20704.232} C_VEL
LIN {X 0,Y 313.331,Z 474.78,A -85,B 0,C 180,E1 20716.977,E2 20716.977} C_VEL
LIN {X 0,Y 329.051,Z 497.399,A -85,B 0,C 180,E1 20726.066,E2 20726.066} C_VEL
LIN {X 0,Y 354.158,Z 537.739,A -85,B 0,C 180,E1 20735.236,E2 20735.236} C_VEL
LIN {X 0,Y 372.185,Z 582.6,A -85,B 0,C 180,E1 20742.176,E2 20742.176} C_VEL
LIN {X 0,Y 375.173,Z 602.924,A -85,B 0,C 180,E1 20744.612,E2 20744.612} C_VEL
LIN {X 0,Y 357.765,Z 658.85,A -85,B 0,C 180,E1 20749.544,E2 20749.544} C_VEL
LIN {X 0,Y 339.019,Z 705.796,A -85,B 0,C 180,E1 20756.773,E2 20756.773} C_VEL
LIN {X 0,Y 323.805,Z 742.052,A -85,B 0,C 180,E1 20766.541,E2 20766.541} C_VEL
LIN {X 0,Y 316.668,Z 763.93,A -85,B 0,C 180,E1 20777.555,E2 20777.555} C_VEL
LIN {X 0,Y 315.309,Z 771.814,A -85,B 0,C 180,E1 20788.622,E2 20788.622} C_VEL
LIN {X 0,Y 315.774,Z 768.35,A -85,B 0,C 180,E1 20798.284,E2 20798.284} C_VEL
LIN {X 0,Y 320.78,Z 750.462,A -85,B 0,C 180,E1 20810.044,E2 20810.044} C_VEL
LIN {X 0,Y 333.513,Z 719.147,A -85,B 0,C 180,E1 20820.237,E2 20820.237} C_VEL
LIN {X 0,Y 351.466,Z 675.508,A -85,B 0,C 180,E1 20828.334,E2 20828.334} C_VEL
LIN {X 0,Y 369.915,Z 622.059,A -85,B 0,C 180,E1 20834.029,E2 20834.029} C_VEL
LIN {X 0,Y 375.465,Z 594.977,A -85,B 0,C 180,E1 20836.155,E2 20836.155} C_VEL
LIN {X 0,Y 358.848,Z 546.969,A -85,B 0,C 180,E1 20843.145,E2 20843.145} C_VEL
LIN {X 0,Y 335.771,Z 506.956,A -85,B 0,C 180,E1 20851.276,E2 20851.276} C_VEL
LIN {X 0,Y 317.034,Z 481.637,A -85,B 0,C 180,E1 20859.742,E2 20859.742} C_VEL
LIN {X 0,Y 313.345,Z 474.78,A -85,B 0,C 180,E1 20863.024,E2 20863.024} C_VEL
LIN {X 0,Y 313.369,Z 474.78,A -85,B 0,C 180,E1 20863.533,E2 20863.533} C_VEL
LIN {X 0,Y 305.904,Z 474.78,A -85,B 0,C 180,E1 20869.994,E2 20869.994} C_VEL
LIN {X 0,Y 306.575,Z 474.78,A -85,B 0,C 180,E1 20881.333,E2 20881.333} C_VEL
LIN {X 0,Y 305.847,Z 476.736,A -85,B 0,C 180,E1 20893.383,E2 20893.383} C_VEL
LIN {X 0,Y 317.656,Z 492.598,A -85,B 0,C 180,E1 20901.541,E2 20901.541} C_VEL
LIN {X 0,Y 338.931,Z 523.559,A -85,B 0,C 180,E1 20910.988,E2 20910.988} C_VEL
LIN {X 0,Y 371.494,Z 578.39,A -85,B 0,C 180,E1 20922.668,E2 20922.668} C_VEL
LIN {X 0,Y 398.146,Z 608.847,A -85,B 0,C 180,E1 20930.473,E2 20930.473} C_VEL
LIN {X 0,Y 421.224,Z 634.792,A -85,B 0,C 180,E1 20938.532,E2 20938.532} C_VEL
LIN {X 0,Y 440.209,Z 654.926,A -85,B 0,C 180,E1 20946.661,E2 20946.661} C_VEL
LIN {X 0,Y 453.12,Z 668.33,A -85,B 0,C 180,E1 20954.184,E2 20954.184} C_VEL
LIN {X 0,Y 459.629,Z 674.585,A -85,B 0,C 180,E1 20959.545,E2 20959.545} C_VEL
LIN {X 0,Y 464.706,Z 678.625,A -85,B 0,C 180,E1 20967.194,E2 20967.194} C_VEL
LIN {X 0,Y 463.777,Z 678.261,A -85,B 0,C 180,E1 20974.689,E2 20974.689} C_VEL
LIN {X 0,Y 457.894,Z 672.069,A -85,B 0,C 180,E1 20982.452,E2 20982.452} C_VEL
LIN {X 0,Y 445.35,Z 660.355,A -85,B 0,C 180,E1 20990.635,E2 20990.635} C_VEL
LIN {X 0,Y 428.558,Z 642.939,A -85,B 0,C 180,E1 20998.536,E2 20998.536} C_VEL
LIN {X 0,Y 406.422,Z 618.92,A -85,B 0,C 180,E1 21006.727,E2 21006.727} C_VEL
LIN {X 0,Y 380.694,Z 589.853,A -85,B 0,C 180,E1 21014.667,E2 21014.667} C_VEL
LIN {X 0,Y 347.858,Z 540.787,A -85,B 0,C 180,E1 21025.433,E2 21025.433} C_VEL
LIN {X 0,Y 325.934,Z 503.39,A -85,B 0,C 180,E1 21034.443,E2 21034.443} C_VEL
LIN {X 0,Y 309.583,Z 481.658,A -85,B 0,C 180,E1 21043.537,E2 21043.537} C_VEL
LIN {X 0,Y 306.048,Z 474.78,A -85,B 0,C 180,E1 21047.197,E2 21047.197} C_VEL
LIN {X 0,Y 306.783,Z 474.78,A -85,B 0,C 180,E1 21058.668,E2 21058.668} C_VEL
LIN {X 0,Y 305.916,Z 474.78,A -85,B 0,C 180,E1 21070.083,E2 21070.083} C_VEL
LIN {X 0,Y 305.997,Z 477.086,A -85,B 0,C 180,E1 21073.23,E2 21073.23} C_VEL
LIN {X 0,Y 317.18,Z 491.847,A -85,B 0,C 180,E1 21080.966,E2 21080.966} C_VEL
LIN {X 0,Y 338.565,Z 522.799,A -85,B 0,C 180,E1 21090.364,E2 21090.364} C_VEL
LIN {X 0,Y 359.775,Z 565.88,A -85,B 0,C 180,E1 21098.48,E2 21098.48} C_VEL
LIN {X 0,Y 369.428,Z 603.318,A -85,B 0,C 180,E1 21103.762,E2 21103.762} C_VEL
LIN {X 0,Y 351.6,Z 658.746,A -85,B 0,C 180,E1 21108.694,E2 21108.694} C_VEL
LIN {X 0,Y 331.563,Z 707.119,A -85,B 0,C 180,E1 21116.319,E2 21116.319} C_VEL
LIN {X 0,Y 316.361,Z 741.874,A -85,B 0,C 180,E1 21125.955,E2 21125.955} C_VEL
LIN {X 0,Y 308.751,Z 763.753,A -85,B 0,C 180,E1 21137.231,E2 21137.231} C_VEL
LIN {X 0,Y 307.306,Z 771.639,A -85,B 0,C 180,E1 21148.586,E2 21148.586} C_VEL
LIN {X 0,Y 307.793,Z 768.3,A -85,B 0,C 180,E1 21158.341,E2 21158.341} C_VEL
LIN {X 0,Y 312.59,Z 751.801,A -85,B 0,C 180,E1 21169.852,E2 21169.852} C_VEL
LIN {X 0,Y 325.559,Z 721.192,A -85,B 0,C 180,E1 21180.407,E2 21180.407} C_VEL
LIN {X 0,Y 344.301,Z 677.456,A -85,B 0,C 180,E1 21188.877,E2 21188.877} C_VEL
LIN {X 0,Y 363.685,Z 623.533,A -85,B 0,C 180,E1 21194.783,E2 21194.783} C_VEL
LIN {X 0,Y 369.341,Z 598.417,A -85,B 0,C 180,E1 21196.767,E2 21196.767} C_VEL
LIN {X 0,Y 354.035,Z 551.833,A -85,B 0,C 180,E1 21203.82,E2 21203.82} C_VEL
LIN {X 0,Y 332.261,Z 512.683,A -85,B 0,C 180,E1 21212.096,E2 21212.096} C_VEL
LIN {X 0,Y 314.33,Z 488.509,A -85,B 0,C 180,E1 21220.645,E2 21220.645} C_VEL
LIN {X 0,Y 307.985,Z 480.59,A -85,B 0,C 180,E1 21224.987,E2 21224.987} C_VEL
LIN {X 0,Y 305.769,Z 474.78,A -85,B 0,C 180,E1 21228.465,E2 21228.465} C_VEL
LIN {X 0,Y 305.904,Z 474.78,A -85,B 0,C 180,E1 21229.994,E2 21229.994} C_VEL
LIN {X 0,Y 298.598,Z 474.785,A -85,B 0,C 180,E1 21236.493,E2 21236.493} C_VEL
LIN {X 0,Y 298.76,Z 477.085,A -85,B 0,C 180,E1 21245.011,E2 21245.011} C_VEL
LIN {X 0,Y 304.784,Z 485.633,A -85,B 0,C 180,E1 21253.431,E2 21253.431} C_VEL
LIN {X 0,Y 315.783,Z 500.072,A -85,B 0,C 180,E1 21261.125,E2 21261.125} C_VEL
LIN {X 0,Y 336.296,Z 531.49,A -85,B 0,C 180,E1 21270.786,E2 21270.786} C_VEL
LIN {X 0,Y 367.272,Z 585.434,A -85,B 0,C 180,E1 21282.667,E2 21282.667} C_VEL
LIN {X 0,Y 394.985,Z 617.282,A -85,B 0,C 180,E1 21290.959,E2 21290.959} C_VEL
LIN {X 0,Y 418.183,Z 643.292,A -85,B 0,C 180,E1 21299.219,E2 21299.219} C_VEL
LIN {X 0,Y 436.067,Z 662.173,A -85,B 0,C 180,E1 21307.069,E2 21307.069} C_VEL
LIN {X 0,Y 448.49,Z 674.848,A -85,B 0,C 180,E1 21314.392,E2 21314.392} C_VEL
LIN {X 0,Y 456.017,Z 682.555,A -85,B 0,C 180,E1 21321.394,E2 21321.394} C_VEL
LIN {X 0,Y 459.8,Z 685.258,A -85,B 0,C 180,E1 21329.055,E2 21329.055} C_VEL
LIN {X 0,Y 457.608,Z 683.599,A -85,B 0,C 180,E1 21336.661,E2 21336.661} C_VEL
LIN {X 0,Y 450.013,Z 675.874,A -85,B 0,C 180,E1 21344.64,E2 21344.64} C_VEL
LIN {X 0,Y 437.775,Z 664.194,A -85,B 0,C 180,E1 21351.992,E2 21351.992} C_VEL
LIN {X 0,Y 420.173,Z 645.789,A -85,B 0,C 180,E1 21359.932,E2 21359.932} C_VEL
LIN {X 0,Y 397.538,Z 620.84,A -85,B 0,C 180,E1 21368.109,E2 21368.109} C_VEL
LIN {X 0,Y 370.694,Z 589.895,A -85,B 0,C 180,E1 21376.292,E2 21376.292} C_VEL
LIN {X 0,Y 340.678,Z 540.436,A -85,B 0,C 180,E1 21387.278,E2 21387.278} C_VEL
LIN {X 0,Y 319.329,Z 504.236,A -85,B 0,C 180,E1 21397.011,E2 21397.011} C_VEL
LIN {X 0,Y 305.996,Z 487.128,A -85,B 0,C 180,E1 21405.5,E2 21405.5} C_VEL
LIN {X 0,Y 302.112,Z 481.71,A -85,B 0,C 180,E1 21409.416,E2 21409.416} C_VEL
LIN {X 0,Y 298.774,Z 474.78,A -85,B 0,C 180,E1 21418.632,E2 21418.632} C_VEL
LIN {X 0,Y 298.915,Z 477.637,A -85,B 0,C 180,E1 21425.183,E2 21425.183} C_VEL
LIN {X 0,Y 304.703,Z 485.41,A -85,B 0,C 180,E1 21433.036,E2 21433.036} C_VEL
LIN {X 0,Y 315.686,Z 500.154,A -85,B 0,C 180,E1 21440.777,E2 21440.777} C_VEL
LIN {X 0,Y 335.321,Z 529.477,A -85,B 0,C 180,E1 21449.845,E2 21449.845} C_VEL
LIN {X 0,Y 354.815,Z 571.187,A -85,B 0,C 180,E1 21457.944,E2 21457.944} C_VEL
LIN {X 0,Y 363.085,Z 606.162,A -85,B 0,C 180,E1 21463.036,E2 21463.036} C_VEL
LIN {X 0,Y 344.487,Z 661.354,A -85,B 0,C 180,E1 21468.141,E2 21468.141} C_VEL
LIN {X 0,Y 324.129,Z 708.442,A -85,B 0,C 180,E1 21475.844,E2 21475.844} C_VEL
LIN {X 0,Y 307.844,Z 744.094,A -85,B 0,C 180,E1 21486.29,E2 21486.29} C_VEL
LIN {X 0,Y 300.488,Z 765.18,A -85,B 0,C 180,E1 21498.354,E2 21498.354} C_VEL
LIN {X 0,Y 299.302,Z 771.464,A -85,B 0,C 180,E1 21508.548,E2 21508.548} C_VEL
LIN {X 0,Y 299.858,Z 767.926,A -85,B 0,C 180,E1 21518.821,E2 21518.821} C_VEL
LIN {X 0,Y 305.46,Z 750.104,A -85,B 0,C 180,E1 21531.096,E2 21531.096} C_VEL
LIN {X 0,Y 319.761,Z 718.143,A -85,B 0,C 180,E1 21541.878,E2 21541.878} C_VEL
LIN {X 0,Y 339.729,Z 673.027,A -85,B 0,C 180,E1 21550.335,E2 21550.335} C_VEL
LIN {X 0,Y 359.592,Z 617.963,A -85,B 0,C 180,E1 21556.106,E2 21556.106} C_VEL
LIN {X 0,Y 363.083,Z 600.867,A -85,B 0,C 180,E1 21557.538,E2 21557.538} C_VEL
LIN {X 0,Y 348.458,Z 554.941,A -85,B 0,C 180,E1 21564.836,E2 21564.836} C_VEL
LIN {X 0,Y 327.608,Z 516.474,A -85,B 0,C 180,E1 21573.44,E2 21573.44} C_VEL
LIN {X 0,Y 308.22,Z 489.601,A -85,B 0,C 180,E1 21584.067,E2 21584.067} C_VEL
LIN {X 0,Y 301.729,Z 481.591,A -85,B 0,C 180,E1 21590.142,E2 21590.142} C_VEL
LIN {X 0,Y 298.598,Z 474.785,A -85,B 0,C 180,E1 21596.493,E2 21596.493} C_VEL
LIN {X 0,Y 297.399,Z 482.705,A -85,B 0,C 180,E1 21603.132,E2 21603.132} C_VEL
LIN {X 0,Y 303.77,Z 494.122,A -85,B 0,C 180,E1 21613.476,E2 21613.476} C_VEL
LIN {X 0,Y 317.202,Z 511.86,A -85,B 0,C 180,E1 21622.594,E2 21622.594} C_VEL
LIN {X 0,Y 336.951,Z 546.765,A -85,B 0,C 180,E1 21632.279,E2 21632.279} C_VEL
LIN {X 0,Y 365.401,Z 595.251,A -85,B 0,C 180,E1 21643.424,E2 21643.424} C_VEL
LIN {X 0,Y 392.028,Z 625.918,A -85,B 0,C 180,E1 21651.61,E2 21651.61} C_VEL
LIN {X 0,Y 414.119,Z 650.725,A -85,B 0,C 180,E1 21659.639,E2 21659.639} C_VEL
LIN {X 0,Y 431.944,Z 669.403,A -85,B 0,C 180,E1 21667.606,E2 21667.606} C_VEL
LIN {X 0,Y 445.474,Z 682.502,A -85,B 0,C 180,E1 21675.846,E2 21675.846} C_VEL
LIN {X 0,Y 452.154,Z 689.77,A -85,B 0,C 180,E1 21683.259,E2 21683.259} C_VEL
LIN {X 0,Y 454.575,Z 691.305,A -85,B 0,C 180,E1 21689.044,E2 21689.044} C_VEL
LIN {X 0,Y 452.29,Z 689.579,A -85,B 0,C 180,E1 21696.739,E2 21696.739} C_VEL
LIN {X 0,Y 444.53,Z 681.726,A -85,B 0,C 180,E1 21704.825,E2 21704.825} C_VEL
LIN {X 0,Y 431.863,Z 669.504,A -85,B 0,C 180,E1 21712.388,E2 21712.388} C_VEL
LIN {X 0,Y 413.521,Z 650.285,A -85,B 0,C 180,E1 21720.557,E2 21720.557} C_VEL
LIN {X 0,Y 391.756,Z 626.195,A -85,B 0,C 180,E1 21728.394,E2 21728.394} C_VEL
LIN {X 0,Y 362.717,Z 592.541,A -85,B 0,C 180,E1 21737.359,E2 21737.359} C_VEL
LIN {X 0,Y 333.689,Z 540.155,A -85,B 0,C 180,E1 21749.246,E2 21749.246} C_VEL
LIN {X 0,Y 314.076,Z 507.846,A -85,B 0,C 180,E1 21759.125,E2 21759.125} C_VEL
LIN {X 0,Y 301.997,Z 490.107,A -85,B 0,C 180,E1 21768.494,E2 21768.494} C_VEL
LIN {X 0,Y 297.079,Z 482.585,A -85,B 0,C 180,E1 21778.624,E2 21778.624} C_VEL
LIN {X 0,Y 298.041,Z 486.139,A -85,B 0,C 180,E1 21785.53,E2 21785.53} C_VEL
LIN {X 0,Y 303.599,Z 493.735,A -85,B 0,C 180,E1 21792.992,E2 21792.992} C_VEL
LIN {X 0,Y 317.185,Z 511.759,A -85,B 0,C 180,E1 21802.217,E2 21802.217} C_VEL
LIN {X 0,Y 338.14,Z 548.031,A -85,B 0,C 180,E1 21812.041,E2 21812.041} C_VEL
LIN {X 0,Y 354.286,Z 591.742,A -85,B 0,C 180,E1 21819.865,E2 21819.865} C_VEL
LIN {X 0,Y 356.602,Z 609.526,A -85,B 0,C 180,E1 21822.333,E2 21822.333} C_VEL
LIN {X 0,Y 336.82,Z 665.506,A -85,B 0,C 180,E1 21827.76,E2 21827.76} C_VEL
LIN {X 0,Y 316.026,Z 711.265,A -85,B 0,C 180,E1 21835.678,E2 21835.678} C_VEL
LIN {X 0,Y 299.554,Z 745.809,A -85,B 0,C 180,E1 21846.437,E2 21846.437} C_VEL
LIN {X 0,Y 292.55,Z 765.003,A -85,B 0,C 180,E1 21858.033,E2 21858.033} C_VEL
LIN {X 0,Y 291.309,Z 771.29,A -85,B 0,C 180,E1 21868.508,E2 21868.508} C_VEL
LIN {X 0,Y 291.89,Z 767.75,A -85,B 0,C 180,E1 21879.063,E2 21879.063} C_VEL
LIN {X 0,Y 297.836,Z 749.925,A -85,B 0,C 180,E1 21891.663,E2 21891.663} C_VEL
LIN {X 0,Y 312.788,Z 718.076,A -85,B 0,C 180,E1 21902.641,E2 21902.641} C_VEL
LIN {X 0,Y 332.993,Z 674.269,A -85,B 0,C 180,E1 21911.037,E2 21911.037} C_VEL
LIN {X 0,Y 353.299,Z 620.232,A -85,B 0,C 180,E1 21916.861,E2 21916.861} C_VEL
LIN {X 0,Y 356.707,Z 602.52,A -85,B 0,C 180,E1 21918.459,E2 21918.459} C_VEL
LIN {X 0,Y 342.487,Z 557.002,A -85,B 0,C 180,E1 21926.093,E2 21926.093} C_VEL
LIN {X 0,Y 323.36,Z 521.376,A -85,B 0,C 180,E1 21934.654,E2 21934.654} C_VEL
LIN {X 0,Y 306.312,Z 496.997,A -85,B 0,C 180,E1 21944.703,E2 21944.703} C_VEL
LIN {X 0,Y 300.032,Z 489.086,A -85,B 0,C 180,E1 21951.003,E2 21951.003} C_VEL
LIN {X 0,Y 297.143,Z 482.588,A -85,B 0,C 180,E1 21958.449,E2 21958.449} C_VEL
LIN {X 0,Y 297.399,Z 482.705,A -85,B 0,C 180,E1 21963.132,E2 21963.132} C_VEL
LIN {X 0,Y 299.057,Z 497.061,A -85,B 0,C 180,E1 21969.325,E2 21969.325} C_VEL
LIN {X 0,Y 307.238,Z 508.613,A -85,B 0,C 180,E1 21977.239,E2 21977.239} C_VEL
LIN {X 0,Y 322.891,Z 533.001,A -85,B 0,C 180,E1 21986.61,E2 21986.61} C_VEL
LIN {X 0,Y 350.196,Z 587.592,A -85,B 0,C 180,E1 21999.728,E2 21999.728} C_VEL
LIN {X 0,Y 383.351,Z 627.866,A -85,B 0,C 180,E1 22010.406,E2 22010.406} C_VEL
LIN {X 0,Y 406.436,Z 653.897,A -85,B 0,C 180,E1 22018.657,E2 22018.657} C_VEL
LIN {X 0,Y 424.91,Z 673.441,A -85,B 0,C 180,E1 22026.73,E2 22026.73} C_VEL
LIN {X 0,Y 438.689,Z 687.353,A -85,B 0,C 180,E1 22034.974,E2 22034.974} C_VEL
LIN {X 0,Y 445.114,Z 694.201,A -85,B 0,C 180,E1 22041.181,E2 22041.181} C_VEL
LIN {X 0,Y 449.032,Z 697.065,A -85,B 0,C 180,E1 22049.033,E2 22049.033} C_VEL
LIN {X 0,Y 446.767,Z 695.348,A -85,B 0,C 180,E1 22056.823,E2 22056.823} C_VEL
LIN {X 0,Y 438.717,Z 687.31,A -85,B 0,C 180,E1 22065.026,E2 22065.026} C_VEL
LIN {X 0,Y 425.806,Z 674.672,A -85,B 0,C 180,E1 22072.738,E2 22072.738} C_VEL
LIN {X 0,Y 407.498,Z 655.451,A -85,B 0,C 180,E1 22080.851,E2 22080.851} C_VEL
LIN {X 0,Y 384.199,Z 629.594,A -85,B 0,C 180,E1 22089.181,E2 22089.181} C_VEL
LIN {X 0,Y 350.952,Z 589.053,A -85,B 0,C 180,E1 22099.951,E2 22099.951} C_VEL
LIN {X 0,Y 322.863,Z 533.127,A -85,B 0,C 180,E1 22113.387,E2 22113.387} C_VEL
LIN {X 0,Y 305.716,Z 505.132,A -85,B 0,C 180,E1 22124.064,E2 22124.064} C_VEL
LIN {X 0,Y 298.483,Z 496.345,A -85,B 0,C 180,E1 22131.501,E2 22131.501} C_VEL
LIN {X 0,Y 296.105,Z 490.525,A -85,B 0,C 180,E1 22138.62,E2 22138.62} C_VEL
LIN {X 0,Y 297.158,Z 494.411,A -85,B 0,C 180,E1 22145.792,E2 22145.792} C_VEL
LIN {X 0,Y 302.412,Z 501.863,A -85,B 0,C 180,E1 22152.86,E2 22152.86} C_VEL
LIN {X 0,Y 315.601,Z 520.436,A -85,B 0,C 180,E1 22162.149,E2 22162.149} C_VEL
LIN {X 0,Y 334.487,Z 554.92,A -85,B 0,C 180,E1 22171.655,E2 22171.655} C_VEL
LIN {X 0,Y 348.827,Z 596.967,A -85,B 0,C 180,E1 22179.425,E2 22179.425} C_VEL
LIN {X 0,Y 350.203,Z 612.432,A -85,B 0,C 180,E1 22181.585,E2 22181.585} C_VEL
LIN {X 0,Y 329.955,Z 667.359,A -85,B 0,C 180,E1 22187.095,E2 22187.095} C_VEL
LIN {X 0,Y 308.499,Z 712.793,A -85,B 0,C 180,E1 22195.22,E2 22195.22} C_VEL
LIN {X 0,Y 291.705,Z 746.529,A -85,B 0,C 180,E1 22206.174,E2 22206.174} C_VEL
LIN {X 0,Y 284.635,Z 764.826,A -85,B 0,C 180,E1 22217.695,E2 22217.695} C_VEL
LIN {X 0,Y 283.305,Z 771.115,A -85,B 0,C 180,E1 22228.466,E2 22228.466} C_VEL
LIN {X 0,Y 283.893,Z 767.759,A -85,B 0,C 180,E1 22239.066,E2 22239.066} C_VEL
LIN {X 0,Y 289.656,Z 751.265,A -85,B 0,C 180,E1 22251.499,E2 22251.499} C_VEL
LIN {X 0,Y 304.672,Z 720.559,A -85,B 0,C 180,E1 22262.772,E2 22262.772} C_VEL
LIN {X 0,Y 325.243,Z 677.977,A -85,B 0,C 180,E1 22271.415,E2 22271.415} C_VEL
LIN {X 0,Y 346.369,Z 624.506,A -85,B 0,C 180,E1 22277.477,E2 22277.477} C_VEL
LIN {X 0,Y 350.685,Z 605.759,A -85,B 0,C 180,E1 22279.179,E2 22279.179} C_VEL
LIN {X 0,Y 337.568,Z 561.522,A -85,B 0,C 180,E1 22286.91,E2 22286.91} C_VEL
LIN {X 0,Y 319.853,Z 526.942,A -85,B 0,C 180,E1 22295.575,E2 22295.575} C_VEL
LIN {X 0,Y 304.289,Z 504.201,A -85,B 0,C 180,E1 22305.475,E2 22305.475} C_VEL
LIN {X 0,Y 298.538,Z 496.608,A -85,B 0,C 180,E1 22311.694,E2 22311.694} C_VEL
LIN {X 0,Y 296.172,Z 490.497,A -85,B 0,C 180,E1 22318.444,E2 22318.444} C_VEL
LIN {X 0,Y 296.833,Z 493.664,A -85,B 0,C 180,E1 22325.268,E2 22325.268} C_VEL
LIN {X 0,Y 299.057,Z 497.061,A -85,B 0,C 180,E1 22329.325,E2 22329.325} C_VEL
LIN {X 0,Y 301.21,Z 510.024,A -85,B 0,C 180,E1 22333.159,E2 22333.159} C_VEL
LIN {X 0,Y 314.088,Z 529.847,A -85,B 0,C 180,E1 22342.831,E2 22342.831} C_VEL
LIN {X 0,Y 330.071,Z 562.51,A -85,B 0,C 180,E1 22352.013,E2 22352.013} C_VEL
LIN {X 0,Y 356.612,Z 609.086,A -85,B 0,C 180,E1 22363.637,E2 22363.637} C_VEL
LIN {X 0,Y 384.951,Z 641.801,A -85,B 0,C 180,E1 22372.784,E2 22372.784} C_VEL
LIN {X 0,Y 406.831,Z 666.127,A -85,B 0,C 180,E1 22381.078,E2 22381.078} C_VEL
LIN {X 0,Y 423.315,Z 683.362,A -85,B 0,C 180,E1 22388.892,E2 22388.892} C_VEL
LIN {X 0,Y 435.8,Z 695.121,A -85,B 0,C 180,E1 22396.927,E2 22396.927} C_VEL
LIN {X 0,Y 442.072,Z 701.799,A -85,B 0,C 180,E1 22405.08,E2 22405.08} C_VEL
LIN {X 0,Y 442.866,Z 702.355,A -85,B 0,C 180,E1 22412.944,E2 22412.944} C_VEL
LIN {X 0,Y 437.694,Z 697.63,A -85,B 0,C 180,E1 22420.986,E2 22420.986} C_VEL
LIN {X 0,Y 427.509,Z 687.458,A -85,B 0,C 180,E1 22428.751,E2 22428.751} C_VEL
LIN {X 0,Y 410.941,Z 670.793,A -85,B 0,C 180,E1 22437.093,E2 22437.093} C_VEL
LIN {X 0,Y 390.202,Z 648.255,A -85,B 0,C 180,E1 22445.277,E2 22445.277} C_VEL
LIN {X 0,Y 364.284,Z 618.983,A -85,B 0,C 180,E1 22453.772,E2 22453.772} C_VEL
LIN {X 0,Y 332.484,Z 569.145,A -85,B 0,C 180,E1 22466.564,E2 22466.564} C_VEL
LIN {X 0,Y 316.438,Z 533.971,A -85,B 0,C 180,E1 22475.757,E2 22475.757} C_VEL
LIN {X 0,Y 302.677,Z 511.582,A -85,B 0,C 180,E1 22485.481,E2 22485.481} C_VEL
LIN {X 0,Y 297.047,Z 503.818,A -85,B 0,C 180,E1 22492.199,E2 22492.199} C_VEL
LIN {X 0,Y 295.131,Z 498.457,A -85,B 0,C 180,E1 22498.615,E2 22498.615} C_VEL
LIN {X 0,Y 296.147,Z 502.412,A -85,B 0,C 180,E1 22505.748,E2 22505.748} C_VEL
LIN {X 0,Y 301.505,Z 510.357,A -85,B 0,C 180,E1 22513.084,E2 22513.084} C_VEL
LIN {X 0,Y 315.943,Z 532.101,A -85,B 0,C 180,E1 22523.336,E2 22523.336} C_VEL
LIN {X 0,Y 333.268,Z 568.153,A -85,B 0,C 180,E1 22532.668,E2 22532.668} C_VEL
LIN {X 0,Y 344.744,Z 609.766,A -85,B 0,C 180,E1 22540.209,E2 22540.209} C_VEL
LIN {X 0,Y 324.563,Z 666.12,A -85,B 0,C 180,E1 22545.971,E2 22545.971} C_VEL
LIN {X 0,Y 301.756,Z 712.741,A -85,B 0,C 180,E1 22554.367,E2 22554.367} C_VEL
LIN {X 0,Y 284.283,Z 746.351,A -85,B 0,C 180,E1 22565.512,E2 22565.512} C_VEL
LIN {X 0,Y 276.734,Z 764.649,A -85,B 0,C 180,E1 22577.338,E2 22577.338} C_VEL
LIN {X 0,Y 275.3,Z 770.94,A -85,B 0,C 180,E1 22588.422,E2 22588.422} C_VEL
LIN {X 0,Y 275.954,Z 767.469,A -85,B 0,C 180,E1 22599.489,E2 22599.489} C_VEL
LIN {X 0,Y 282.071,Z 751.087,A -85,B 0,C 180,E1 22612.107,E2 22612.107} C_VEL
LIN {X 0,Y 297.824,Z 720.381,A -85,B 0,C 180,E1 22623.624,E2 22623.624} C_VEL
LIN {X 0,Y 319.523,Z 677.061,A -85,B 0,C 180,E1 22632.488,E2 22632.488} C_VEL
LIN {X 0,Y 341.492,Z 622.92,A -85,B 0,C 180,E1 22638.595,E2 22638.595} C_VEL
LIN {X 0,Y 344.619,Z 608.42,A -85,B 0,C 180,E1 22640.001,E2 22640.001} C_VEL
LIN {X 0,Y 332.344,Z 565.226,A -85,B 0,C 180,E1 22647.893,E2 22647.893} C_VEL
LIN {X 0,Y 315.522,Z 531.352,A -85,B 0,C 180,E1 22656.912,E2 22656.912} C_VEL
LIN {X 0,Y 301.424,Z 510.266,A -85,B 0,C 180,E1 22667.005,E2 22667.005} C_VEL
LIN {X 0,Y 296.236,Z 502.663,A -85,B 0,C 180,E1 22674.032,E2 22674.032} C_VEL
LIN {X 0,Y 295.199,Z 498.423,A -85,B 0,C 180,E1 22678.439,E2 22678.439} C_VEL
LIN {X 0,Y 295.835,Z 501.678,A -85,B 0,C 180,E1 22685.245,E2 22685.245} C_VEL
LIN {X 0,Y 301.21,Z 510.024,A -85,B 0,C 180,E1 22693.159,E2 22693.159} C_VEL
LIN {X 0,Y 306.405,Z 528.05,A -85,B 0,C 180,E1 22698.858,E2 22698.858} C_VEL
LIN {X 0,Y 321.961,Z 558.401,A -85,B 0,C 180,E1 22709.063,E2 22709.063} C_VEL
LIN {X 0,Y 346.473,Z 609.046,A -85,B 0,C 180,E1 22721.797,E2 22721.797} C_VEL
LIN {X 0,Y 377.871,Z 645.836,A -85,B 0,C 180,E1 22732.298,E2 22732.298} C_VEL
LIN {X 0,Y 400.297,Z 670.87,A -85,B 0,C 180,E1 22740.773,E2 22740.773} C_VEL
LIN {X 0,Y 417.552,Z 688.877,A -85,B 0,C 180,E1 22748.934,E2 22748.934} C_VEL
LIN {X 0,Y 429.603,Z 700.286,A -85,B 0,C 180,E1 22756.736,E2 22756.736} C_VEL
LIN {X 0,Y 436.109,Z 707.173,A -85,B 0,C 180,E1 22765.013,E2 22765.013} C_VEL
LIN {X 0,Y 437.348,Z 708.079,A -85,B 0,C 180,E1 22770.993,E2 22770.993} C_VEL
LIN {X 0,Y 433.307,Z 704.826,A -85,B 0,C 180,E1 22779.061,E2 22779.061} C_VEL
LIN {X 0,Y 426.483,Z 697.82,A -85,B 0,C 180,E1 22785.467,E2 22785.467} C_VEL
LIN {X 0,Y 413.088,Z 684.418,A -85,B 0,C 180,E1 22793.36,E2 22793.36} C_VEL
LIN {X 0,Y 394.383,Z 664.684,A -85,B 0,C 180,E1 22801.581,E2 22801.581} C_VEL
LIN {X 0,Y 370.475,Z 638.034,A -85,B 0,C 180,E1 22810.075,E2 22810.075} C_VEL
LIN {X 0,Y 332.851,Z 586.709,A -85,B 0,C 180,E1 22824.219,E2 22824.219} C_VEL
LIN {X 0,Y 315.014,Z 543.874,A -85,B 0,C 180,E1 22835.201,E2 22835.201} C_VEL
LIN {X 0,Y 301.187,Z 519.359,A -85,B 0,C 180,E1 22845.687,E2 22845.687} C_VEL
LIN {X 0,Y 294.901,Z 510.151,A -85,B 0,C 180,E1 22854.183,E2 22854.183} C_VEL
LIN {X 0,Y 294.117,Z 506.392,A -85,B 0,C 180,E1 22858.611,E2 22858.611} C_VEL
LIN {X 0,Y 295.203,Z 510.786,A -85,B 0,C 180,E1 22866.174,E2 22866.174} C_VEL
LIN {X 0,Y 302.49,Z 521.097,A -85,B 0,C 180,E1 22875.078,E2 22875.078} C_VEL
LIN {X 0,Y 317.688,Z 548.199,A -85,B 0,C 180,E1 22885.67,E2 22885.67} C_VEL
LIN {X 0,Y 332.347,Z 584.838,A -85,B 0,C 180,E1 22894.355,E2 22894.355} C_VEL
LIN {X 0,Y 338.116,Z 616.755,A -85,B 0,C 180,E1 22899.897,E2 22899.897} C_VEL
LIN {X 0,Y 316.255,Z 671.256,A -85,B 0,C 180,E1 22905.71,E2 22905.71} C_VEL
LIN {X 0,Y 293.117,Z 716.208,A -85,B 0,C 180,E1 22914.406,E2 22914.406} C_VEL
LIN {X 0,Y 275.94,Z 747.87,A -85,B 0,C 180,E1 22925.658,E2 22925.658} C_VEL
LIN {X 0,Y 268.369,Z 766.057,A -85,B 0,C 180,E1 22938.593,E2 22938.593} C_VEL
LIN {X 0,Y 267.748,Z 770.775,A -85,B 0,C 180,E1 22951.623,E2 22951.623} C_VEL
LIN {X 0,Y 269.328,Z 762.866,A -85,B 0,C 180,E1 22964.677,E2 22964.677} C_VEL
LIN {X 0,Y 279.55,Z 740.982,A -85,B 0,C 180,E1 22977.458,E2 22977.458} C_VEL
LIN {X 0,Y 299.026,Z 705.316,A -85,B 0,C 180,E1 22988.226,E2 22988.226} C_VEL
LIN {X 0,Y 322.293,Z 657.699,A -85,B 0,C 180,E1 22996.096,E2 22996.096} C_VEL
LIN {X 0,Y 338.607,Z 611.706,A -85,B 0,C 180,E1 23000.725,E2 23000.725} C_VEL
LIN {X 0,Y 327.732,Z 570.399,A -85,B 0,C 180,E1 23008.597,E2 23008.597} C_VEL
LIN {X 0,Y 312.26,Z 537.622,A -85,B 0,C 180,E1 23017.695,E2 23017.695} C_VEL
LIN {X 0,Y 298.014,Z 513.625,A -85,B 0,C 180,E1 23029.647,E2 23029.647} C_VEL
LIN {X 0,Y 294.198,Z 506.362,A -85,B 0,C 180,E1 23038.434,E2 23038.434} C_VEL
LIN {X 0,Y 294.777,Z 509.93,A -85,B 0,C 180,E1 23045.449,E2 23045.449} C_VEL
LIN {X 0,Y 302.228,Z 520.782,A -85,B 0,C 180,E1 23055.285,E2 23055.285} C_VEL
LIN {X 0,Y 306.405,Z 528.05,A -85,B 0,C 180,E1 23058.858,E2 23058.858} C_VEL
LIN {X 0,Y 311.274,Z 549.823,A -85,B 0,C 180,E1 23064.017,E2 23064.017} C_VEL
LIN {X 0,Y 325.189,Z 585.616,A -85,B 0,C 180,E1 23073.66,E2 23073.66} C_VEL
LIN {X 0,Y 358.267,Z 635.48,A -85,B 0,C 180,E1 23087.717,E2 23087.717} C_VEL
LIN {X 0,Y 382.595,Z 663.316,A -85,B 0,C 180,E1 23096.152,E2 23096.152} C_VEL
LIN {X 0,Y 402.278,Z 684.664,A -85,B 0,C 180,E1 23104.309,E2 23104.309} C_VEL
LIN {X 0,Y 416.499,Z 699.327,A -85,B 0,C 180,E1 23111.972,E2 23111.972} C_VEL
LIN {X 0,Y 426.084,Z 708.701,A -85,B 0,C 180,E1 23119.574,E2 23119.574} C_VEL
LIN {X 0,Y 431.017,Z 712.706,A -85,B 0,C 180,E1 23126.975,E2 23126.975} C_VEL
LIN {X 0,Y 429.974,Z 712.158,A -85,B 0,C 180,E1 23135.059,E2 23135.059} C_VEL
LIN {X 0,Y 423.173,Z 705.263,A -85,B 0,C 180,E1 23143.47,E2 23143.47} C_VEL
LIN {X 0,Y 410.711,Z 693.479,A -85,B 0,C 180,E1 23151.415,E2 23151.415} C_VEL
LIN {X 0,Y 393.93,Z 675.944,A -85,B 0,C 180,E1 23159.339,E2 23159.339} C_VEL
LIN {X 0,Y 371.231,Z 650.912,A -85,B 0,C 180,E1 23167.86,E2 23167.86} C_VEL
LIN {X 0,Y 332.725,Z 601.865,A -85,B 0,C 180,E1 23182.104,E2 23182.104} C_VEL
LIN {X 0,Y 311.983,Z 551.265,A -85,B 0,C 180,E1 23195.493,E2 23195.493} C_VEL
LIN {X 0,Y 299.146,Z 526.84,A -85,B 0,C 180,E1 23206.056,E2 23206.056} C_VEL
LIN {X 0,Y 293.014,Z 514.318,A -85,B 0,C 180,E1 23217.863,E2 23217.863} C_VEL
LIN {X 0,Y 293.557,Z 517.831,A -85,B 0,C 180,E1 23225.093,E2 23225.093} C_VEL
LIN {X 0,Y 300.372,Z 528.475,A -85,B 0,C 180,E1 23234.625,E2 23234.625} C_VEL
LIN {X 0,Y 314.521,Z 555.249,A -85,B 0,C 180,E1 23245.286,E2 23245.286} C_VEL
LIN {X 0,Y 328.033,Z 592.272,A -85,B 0,C 180,E1 23254.207,E2 23254.207} C_VEL
LIN {X 0,Y 331.956,Z 619.616,A -85,B 0,C 180,E1 23259.062,E2 23259.062} C_VEL
LIN {X 0,Y 309.343,Z 673.491,A -85,B 0,C 180,E1 23265.013,E2 23265.013} C_VEL
LIN {X 0,Y 285.766,Z 717.36,A -85,B 0,C 180,E1 23273.816,E2 23273.816} C_VEL
LIN {X 0,Y 267.696,Z 749.21,A -85,B 0,C 180,E1 23285.75,E2 23285.75} C_VEL
LIN {X 0,Y 260.44,Z 765.88,A -85,B 0,C 180,E1 23298.241,E2 23298.241} C_VEL
LIN {X 0,Y 259.747,Z 770.6,A -85,B 0,C 180,E1 23311.673,E2 23311.673} C_VEL
LIN {X 0,Y 261.483,Z 762.689,A -85,B 0,C 180,E1 23325.128,E2 23325.128} C_VEL
LIN {X 0,Y 273.471,Z 739.009,A -85,B 0,C 180,E1 23339.026,E2 23339.026} C_VEL
LIN {X 0,Y 294.751,Z 701.548,A -85,B 0,C 180,E1 23350.025,E2 23350.025} C_VEL
LIN {X 0,Y 318.96,Z 652.66,A -85,B 0,C 180,E1 23357.742,E2 23357.742} C_VEL
LIN {X 0,Y 332.659,Z 615.16,A -85,B 0,C 180,E1 23361.449,E2 23361.449} C_VEL
LIN {X 0,Y 322.77,Z 574.688,A -85,B 0,C 180,E1 23369.541,E2 23369.541} C_VEL
LIN {X 0,Y 308.783,Z 543.635,A -85,B 0,C 180,E1 23378.569,E2 23378.569} C_VEL
LIN {X 0,Y 296.477,Z 521.393,A -85,B 0,C 180,E1 23389.965,E2 23389.965} C_VEL
LIN {X 0,Y 293.034,Z 514.247,A -85,B 0,C 180,E1 23398.428,E2 23398.428} C_VEL
LIN {X 0,Y 293.697,Z 518.224,A -85,B 0,C 180,E1 23405.841,E2 23405.841} C_VEL
LIN {X 0,Y 300.176,Z 528.635,A -85,B 0,C 180,E1 23415.017,E2 23415.017} C_VEL
LIN {X 0,Y 311.274,Z 549.823,A -85,B 0,C 180,E1 23424.017,E2 23424.017} C_VEL
LIN {X 0,Y 314.782,Z 573.881,A -85,B 0,C 180,E1 23428.806,E2 23428.806} C_VEL
LIN {X 0,Y 336.094,Z 621.213,A -85,B 0,C 180,E1 23441.644,E2 23441.644} C_VEL
LIN {X 0,Y 368.943,Z 660.008,A -85,B 0,C 180,E1 23453.416,E2 23453.416} C_VEL
LIN {X 0,Y 390.456,Z 683.692,A -85,B 0,C 180,E1 23461.811,E2 23461.811} C_VEL
LIN {X 0,Y 406.763,Z 700.554,A -85,B 0,C 180,E1 23469.84,E2 23469.84} C_VEL
LIN {X 0,Y 417.949,Z 711.221,A -85,B 0,C 180,E1 23477.426,E2 23477.426} C_VEL
LIN {X 0,Y 423.481,Z 717.093,A -85,B 0,C 180,E1 23484.864,E2 23484.864} C_VEL
LIN {X 0,Y 424.811,Z 718.026,A -85,B 0,C 180,E1 23491.023,E2 23491.023} C_VEL
LIN {X 0,Y 421.319,Z 715.277,A -85,B 0,C 180,E1 23498.418,E2 23498.418} C_VEL
LIN {X 0,Y 415.175,Z 708.766,A -85,B 0,C 180,E1 23504.688,E2 23504.688} C_VEL
LIN {X 0,Y 402.168,Z 696.11,A -85,B 0,C 180,E1 23512.608,E2 23512.608} C_VEL
LIN {X 0,Y 383.746,Z 676.768,A -85,B 0,C 180,E1 23520.929,E2 23520.929} C_VEL
LIN {X 0,Y 360.41,Z 650.829,A -85,B 0,C 180,E1 23529.446,E2 23529.446} C_VEL
LIN {X 0,Y 322.998,Z 598.495,A -85,B 0,C 180,E1 23544.97,E2 23544.97} C_VEL
LIN {X 0,Y 308.079,Z 557.029,A -85,B 0,C 180,E1 23556.308,E2 23556.308} C_VEL
LIN {X 0,Y 296.795,Z 533.979,A -85,B 0,C 180,E1 23566.697,E2 23566.697} C_VEL
LIN {X 0,Y 291.677,Z 522.17,A -85,B 0,C 180,E1 23578.599,E2 23578.599} C_VEL
LIN {X 0,Y 292.844,Z 527.405,A -85,B 0,C 180,E1 23586.971,E2 23586.971} C_VEL
LIN {X 0,Y 299.473,Z 539.002,A -85,B 0,C 180,E1 23595.61,E2 23595.61} C_VEL
LIN {X 0,Y 311.909,Z 564.282,A -85,B 0,C 180,E1 23605.502,E2 23605.502} C_VEL
LIN {X 0,Y 323.817,Z 601.416,A -85,B 0,C 180,E1 23614.471,E2 23614.471} C_VEL
LIN {X 0,Y 325.751,Z 622.836,A -85,B 0,C 180,E1 23618.235,E2 23618.235} C_VEL
LIN {X 0,Y 302.113,Z 676.482,A -85,B 0,C 180,E1 23624.397,E2 23624.397} C_VEL
LIN {X 0,Y 277.721,Z 719.843,A -85,B 0,C 180,E1 23633.571,E2 23633.571} C_VEL
LIN {X 0,Y 259.24,Z 751.004,A -85,B 0,C 180,E1 23646.103,E2 23646.103} C_VEL
LIN {X 0,Y 252.15,Z 766.941,A -85,B 0,C 180,E1 23659.605,E2 23659.605} C_VEL
LIN {X 0,Y 251.733,Z 770.425,A -85,B 0,C 180,E1 23671.726,E2 23671.726} C_VEL
LIN {X 0,Y 253.672,Z 762.512,A -85,B 0,C 180,E1 23685.606,E2 23685.606} C_VEL
LIN {X 0,Y 266.391,Z 738.831,A -85,B 0,C 180,E1 23699.875,E2 23699.875} C_VEL
LIN {X 0,Y 288.569,Z 701.371,A -85,B 0,C 180,E1 23711.064,E2 23711.064} C_VEL
LIN {X 0,Y 313.522,Z 652.529,A -85,B 0,C 180,E1 23718.837,E2 23718.837} C_VEL
LIN {X 0,Y 326.525,Z 617.164,A -85,B 0,C 180,E1 23722.476,E2 23722.476} C_VEL
LIN {X 0,Y 317.102,Z 577.103,A -85,B 0,C 180,E1 23730.943,E2 23730.943} C_VEL
LIN {X 0,Y 304.041,Z 546.994,A -85,B 0,C 180,E1 23740.415,E2 23740.415} C_VEL
LIN {X 0,Y 294.067,Z 528.709,A -85,B 0,C 180,E1 23751.006,E2 23751.006} C_VEL
LIN {X 0,Y 291.771,Z 522.151,A -85,B 0,C 180,E1 23758.421,E2 23758.421} C_VEL
LIN {X 0,Y 292.228,Z 526.409,A -85,B 0,C 180,E1 23766.058,E2 23766.058} C_VEL
LIN {X 0,Y 298.196,Z 536.812,A -85,B 0,C 180,E1 23774.93,E2 23774.93} C_VEL
LIN {X 0,Y 310.017,Z 561.5,A -85,B 0,C 180,E1 23785.184,E2 23785.184} C_VEL
LIN {X 0,Y 314.782,Z 573.881,A -85,B 0,C 180,E1 23788.806,E2 23788.806} C_VEL
LIN {X 0,Y 316.139,Z 599.297,A -85,B 0,C 180,E1 23793.306,E2 23793.306} C_VEL
LIN {X 0,Y 348.644,Z 648.887,A -85,B 0,C 180,E1 23808.535,E2 23808.535} C_VEL
LIN {X 0,Y 373.571,Z 677.141,A -85,B 0,C 180,E1 23817.513,E2 23817.513} C_VEL
LIN {X 0,Y 393.448,Z 698.097,A -85,B 0,C 180,E1 23826.127,E2 23826.127} C_VEL
LIN {X 0,Y 406.249,Z 711.498,A -85,B 0,C 180,E1 23833.742,E2 23833.742} C_VEL
LIN {X 0,Y 413.9,Z 719.086,A -85,B 0,C 180,E1 23840.51,E2 23840.51} C_VEL
LIN {X 0,Y 418.149,Z 722.265,A -85,B 0,C 180,E1 23846.882,E2 23846.882} C_VEL
LIN {X 0,Y 417.031,Z 721.617,A -85,B 0,C 180,E1 23855.216,E2 23855.216} C_VEL
LIN {X 0,Y 409.759,Z 714.35,A -85,B 0,C 180,E1 23863.92,E2 23863.92} C_VEL
LIN {X 0,Y 396.606,Z 701.725,A -85,B 0,C 180,E1 23872.118,E2 23872.118} C_VEL
LIN {X 0,Y 378.238,Z 682.532,A -85,B 0,C 180,E1 23880.546,E2 23880.546} C_VEL
LIN {X 0,Y 354.979,Z 656.772,A -85,B 0,C 180,E1 23889.131,E2 23889.131} C_VEL
LIN {X 0,Y 317.869,Z 604.179,A -85,B 0,C 180,E1 23905.385,E2 23905.385} C_VEL
LIN {X 0,Y 304.564,Z 563.781,A -85,B 0,C 180,E1 23916.762,E2 23916.762} C_VEL
LIN {X 0,Y 294.406,Z 541.298,A -85,B 0,C 180,E1 23927.155,E2 23927.155} C_VEL
LIN {X 0,Y 290.026,Z 529.988,A -85,B 0,C 180,E1 23938.591,E2 23938.591} C_VEL
LIN {X 0,Y 292.879,Z 537.42,A -85,B 0,C 180,E1 23949.783,E2 23949.783} C_VEL
LIN {X 0,Y 303.872,Z 560.232,A -85,B 0,C 180,E1 23961.506,E2 23961.506} C_VEL
LIN {X 0,Y 315.491,Z 593.045,A -85,B 0,C 180,E1 23970.907,E2 23970.907} C_VEL
LIN {X 0,Y 320.354,Z 623.812,A -85,B 0,C 180,E1 23977.204,E2 23977.204} C_VEL
LIN {X 0,Y 295.772,Z 677.715,A -85,B 0,C 180,E1 23983.498,E2 23983.498} C_VEL
LIN {X 0,Y 270.426,Z 720.996,A -85,B 0,C 180,E1 23992.927,E2 23992.927} C_VEL
LIN {X 0,Y 251.635,Z 751.113,A -85,B 0,C 180,E1 24005.513,E2 24005.513} C_VEL
LIN {X 0,Y 244.218,Z 766.765,A -85,B 0,C 180,E1 24019.264,E2 24019.264} C_VEL
LIN {X 0,Y 243.719,Z 770.249,A -85,B 0,C 180,E1 24031.783,E2 24031.783} C_VEL
LIN {X 0,Y 245.864,Z 762.334,A -85,B 0,C 180,E1 24046.114,E2 24046.114} C_VEL
LIN {X 0,Y 259.322,Z 738.712,A -85,B 0,C 180,E1 24060.746,E2 24060.746} C_VEL
LIN {X 0,Y 282.472,Z 701.192,A -85,B 0,C 180,E1 24072.15,E2 24072.15} C_VEL
LIN {X 0,Y 308.265,Z 652.353,A -85,B 0,C 180,E1 24079.967,E2 24079.967} C_VEL
LIN {X 0,Y 320.594,Z 619.821,A -85,B 0,C 180,E1 24083.414,E2 24083.414} C_VEL
LIN {X 0,Y 312.075,Z 580.99,A -85,B 0,C 180,E1 24092.005,E2 24092.005} C_VEL
LIN {X 0,Y 300.117,Z 552.409,A -85,B 0,C 180,E1 24101.69,E2 24101.69} C_VEL
LIN {X 0,Y 291.798,Z 536.055,A -85,B 0,C 180,E1 24111.877,E2 24111.877} C_VEL
LIN {X 0,Y 290.122,Z 529.96,A -85,B 0,C 180,E1 24118.412,E2 24118.412} C_VEL
LIN {X 0,Y 291.59,Z 535.977,A -85,B 0,C 180,E1 24128.325,E2 24128.325} C_VEL
LIN {X 0,Y 299.749,Z 552.643,A -85,B 0,C 180,E1 24138.843,E2 24138.843} C_VEL
LIN {X 0,Y 310.966,Z 581.599,A -85,B 0,C 180,E1 24148.708,E2 24148.708} C_VEL
LIN {X 0,Y 316.139,Z 599.297,A -85,B 0,C 180,E1 24153.306,E2 24153.306} C_VEL
LIN {X 0,Y 318.748,Z 622.471,A -85,B 0,C 180,E1 24158.129,E2 24158.129} C_VEL
LIN {X 0,Y 355.307,Z 668.573,A -85,B 0,C 180,E1 24173.173,E2 24173.173} C_VEL
LIN {X 0,Y 376.846,Z 692.358,A -85,B 0,C 180,E1 24181.597,E2 24181.597} C_VEL
LIN {X 0,Y 393.173,Z 709.257,A -85,B 0,C 180,E1 24189.62,E2 24189.62} C_VEL
LIN {X 0,Y 405.381,Z 720.975,A -85,B 0,C 180,E1 24198.127,E2 24198.127} C_VEL
LIN {X 0,Y 411.394,Z 726.576,A -85,B 0,C 180,E1 24206.83,E2 24206.83} C_VEL
LIN {X 0,Y 411.143,Z 726.655,A -85,B 0,C 180,E1 24213.172,E2 24213.172} C_VEL
LIN {X 0,Y 406.304,Z 722.248,A -85,B 0,C 180,E1 24220.756,E2 24220.756} C_VEL
LIN {X 0,Y 395.487,Z 711.518,A -85,B 0,C 180,E1 24229.022,E2 24229.022} C_VEL
LIN {X 0,Y 378.996,Z 694.846,A -85,B 0,C 180,E1 24237.397,E2 24237.397} C_VEL
LIN {X 0,Y 358.478,Z 672.693,A -85,B 0,C 180,E1 24245.564,E2 24245.564} C_VEL
LIN {X 0,Y 322.351,Z 629.054,A -85,B 0,C 180,E1 24259.83,E2 24259.83} C_VEL
LIN {X 0,Y 301.336,Z 571.617,A -85,B 0,C 180,E1 24276.826,E2 24276.826} C_VEL
LIN {X 0,Y 292.006,Z 548.766,A -85,B 0,C 180,E1 24287.429,E2 24287.429} C_VEL
LIN {X 0,Y 288.366,Z 537.798,A -85,B 0,C 180,E1 24298.583,E2 24298.583} C_VEL
LIN {X 0,Y 290.832,Z 545.873,A -85,B 0,C 180,E1 24309.961,E2 24309.961} C_VEL
LIN {X 0,Y 300.25,Z 566.56,A -85,B 0,C 180,E1 24320.87,E2 24320.87} C_VEL
LIN {X 0,Y 310.724,Z 599.228,A -85,B 0,C 180,E1 24330.5,E2 24330.5} C_VEL
LIN {X 0,Y 314.053,Z 627.154,A -85,B 0,C 180,E1 24336.34,E2 24336.34} C_VEL
LIN {X 0,Y 288.947,Z 679.781,A -85,B 0,C 180,E1 24342.713,E2 24342.713} C_VEL
LIN {X 0,Y 263.046,Z 722.184,A -85,B 0,C 180,E1 24352.288,E2 24352.288} C_VEL
LIN {X 0,Y 243.802,Z 751.718,A -85,B 0,C 180,E1 24365.179,E2 24365.179} C_VEL
LIN {X 0,Y 236.291,Z 766.588,A -85,B 0,C 180,E1 24378.899,E2 24378.899} C_VEL
LIN {X 0,Y 235.707,Z 770.074,A -85,B 0,C 180,E1 24391.843,E2 24391.843} C_VEL
LIN {X 0,Y 238.085,Z 762.157,A -85,B 0,C 180,E1 24406.656,E2 24406.656} C_VEL
LIN {X 0,Y 252.235,Z 738.694,A -85,B 0,C 180,E1 24421.623,E2 24421.623} C_VEL
LIN {X 0,Y 276.496,Z 701.015,A -85,B 0,C 180,E1 24433.281,E2 24433.281} C_VEL
LIN {X 0,Y 303.375,Z 651.682,A -85,B 0,C 180,E1 24441.198,E2 24441.198} C_VEL
LIN {X 0,Y 314.737,Z 622.758,A -85,B 0,C 180,E1 24444.325,E2 24444.325} C_VEL
LIN {X 0,Y 307.1,Z 584.961,A -85,B 0,C 180,E1 24453.109,E2 24453.109} C_VEL
LIN {X 0,Y 296.33,Z 557.345,A -85,B 0,C 180,E1 24463.077,E2 24463.077} C_VEL
LIN {X 0,Y 289.117,Z 542.933,A -85,B 0,C 180,E1 24473.318,E2 24473.318} C_VEL
LIN {X 0,Y 288.346,Z 537.883,A -85,B 0,C 180,E1 24481.417,E2 24481.417} C_VEL
LIN {X 0,Y 293.039,Z 551.264,A -85,B 0,C 180,E1 24494.05,E2 24494.05} C_VEL
LIN {X 0,Y 302.929,Z 575.982,A -85,B 0,C 180,E1 24504.706,E2 24504.706} C_VEL
LIN {X 0,Y 318.748,Z 622.471,A -85,B 0,C 180,E1 24518.129,E2 24518.129} C_VEL
LIN {X 0,Y 323.296,Z 643.487,A -85,B 0,C 180,E1 24523.163,E2 24523.163} C_VEL
LIN {X 0,Y 354.711,Z 679.732,A -85,B 0,C 180,E1 24535.438,E2 24535.438} C_VEL
LIN {X 0,Y 374.939,Z 701.858,A -85,B 0,C 180,E1 24543.846,E2 24543.846} C_VEL
LIN {X 0,Y 390.236,Z 717.521,A -85,B 0,C 180,E1 24552.06,E2 24552.06} C_VEL
LIN {X 0,Y 399.282,Z 726.144,A -85,B 0,C 180,E1 24559.053,E2 24559.053} C_VEL
LIN {X 0,Y 404.511,Z 730.677,A -85,B 0,C 180,E1 24566.776,E2 24566.776} C_VEL
LIN {X 0,Y 404.245,Z 730.749,A -85,B 0,C 180,E1 24573.226,E2 24573.226} C_VEL
LIN {X 0,Y 399.303,Z 726.179,A -85,B 0,C 180,E1 24580.947,E2 24580.947} C_VEL
LIN {X 0,Y 387.972,Z 715.042,A -85,B 0,C 180,E1 24589.405,E2 24589.405} C_VEL
LIN {X 0,Y 372.436,Z 699.331,A -85,B 0,C 180,E1 24597.247,E2 24597.247} C_VEL
LIN {X 0,Y 351.502,Z 676.744,A -85,B 0,C 180,E1 24605.622,E2 24605.622} C_VEL
LIN {X 0,Y 314.837,Z 631.392,A -85,B 0,C 180,E1 24621.06,E2 24621.06} C_VEL
LIN {X 0,Y 297.216,Z 577.362,A -85,B 0,C 180,E1 24637.584,E2 24637.584} C_VEL
LIN {X 0,Y 289.644,Z 556.567,A -85,B 0,C 180,E1 24647.421,E2 24647.421} C_VEL
LIN {X 0,Y 286.22,Z 545.621,A -85,B 0,C 180,E1 24660.091,E2 24660.091} C_VEL
LIN {X 0,Y 290.276,Z 557.296,A -85,B 0,C 180,E1 24672.543,E2 24672.543} C_VEL
LIN {X 0,Y 299.843,Z 582.267,A -85,B 0,C 180,E1 24683.578,E2 24683.578} C_VEL
LIN {X 0,Y 307.856,Z 616.584,A -85,B 0,C 180,E1 24692.757,E2 24692.757} C_VEL
LIN {X 0,Y 307.517,Z 631.415,A -85,B 0,C 180,E1 24695.543,E2 24695.543} C_VEL
LIN {X 0,Y 281.289,Z 683.391,A -85,B 0,C 180,E1 24702.158,E2 24702.158} C_VEL
LIN {X 0,Y 254.293,Z 725.389,A -85,B 0,C 180,E1 24712.319,E2 24712.319} C_VEL
LIN {X 0,Y 234.76,Z 754.158,A -85,B 0,C 180,E1 24726.188,E2 24726.188} C_VEL
LIN {X 0,Y 227.978,Z 767.54,A -85,B 0,C 180,E1 24740.427,E2 24740.427} C_VEL
LIN {X 0,Y 227.692,Z 769.899,A -85,B 0,C 180,E1 24751.908,E2 24751.908} C_VEL
LIN {X 0,Y 230.328,Z 761.98,A -85,B 0,C 180,E1 24767.234,E2 24767.234} C_VEL
LIN {X 0,Y 244.994,Z 738.959,A -85,B 0,C 180,E1 24782.412,E2 24782.412} C_VEL
LIN {X 0,Y 269.622,Z 702.34,A -85,B 0,C 180,E1 24794.109,E2 24794.109} C_VEL
LIN {X 0,Y 296.831,Z 654.499,A -85,B 0,C 180,E1 24802.045,E2 24802.045} C_VEL
LIN {X 0,Y 308.899,Z 626.46,A -85,B 0,C 180,E1 24805.079,E2 24805.079} C_VEL
LIN {X 0,Y 302.746,Z 590.855,A -85,B 0,C 180,E1 24813.712,E2 24813.712} C_VEL
LIN {X 0,Y 292.84,Z 563.283,A -85,B 0,C 180,E1 24823.976,E2 24823.976} C_VEL
LIN {X 0,Y 286.717,Z 550.139,A -85,B 0,C 180,E1 24834.024,E2 24834.024} C_VEL
LIN {X 0,Y 286.24,Z 545.792,A -85,B 0,C 180,E1 24841.618,E2 24841.618} C_VEL
LIN {X 0,Y 290.151,Z 558.186,A -85,B 0,C 180,E1 24853.517,E2 24853.517} C_VEL
LIN {X 0,Y 298.987,Z 582.528,A -85,B 0,C 180,E1 24864.254,E2 24864.254} C_VEL
LIN {X 0,Y 317.986,Z 636.195,A -85,B 0,C 180,E1 24880.605,E2 24880.605} C_VEL
LIN {X 0,Y 323.296,Z 643.487,A -85,B 0,C 180,E1 24883.163,E2 24883.163} C_VEL
LIN {X 0,Y 329.218,Z 663.012,A -85,B 0,C 180,E1 24888.283,E2 24888.283} C_VEL
LIN {X 0,Y 357.05,Z 694.06,A -85,B 0,C 180,E1 24899.107,E2 24899.107} C_VEL
LIN {X 0,Y 375.288,Z 713.148,A -85,B 0,C 180,E1 24907.426,E2 24907.426} C_VEL
LIN {X 0,Y 387.906,Z 725.859,A -85,B 0,C 180,E1 24915.279,E2 24915.279} C_VEL
LIN {X 0,Y 394.592,Z 732.733,A -85,B 0,C 180,E1 24922.27,E2 24922.27} C_VEL
LIN {X 0,Y 397.83,Z 734.971,A -85,B 0,C 180,E1 24928.908,E2 24928.908} C_VEL
LIN {X 0,Y 396.227,Z 733.843,A -85,B 0,C 180,E1 24935.491,E2 24935.491} C_VEL
LIN {X 0,Y 389.611,Z 727.217,A -85,B 0,C 180,E1 24943.491,E2 24943.491} C_VEL
LIN {X 0,Y 376.541,Z 714.677,A -85,B 0,C 180,E1 24951.812,E2 24951.812} C_VEL
LIN {X 0,Y 358.024,Z 695.361,A -85,B 0,C 180,E1 24960.423,E2 24960.423} C_VEL
LIN {X 0,Y 330.78,Z 665.472,A -85,B 0,C 180,E1 24970.936,E2 24970.936} C_VEL
LIN {X 0,Y 301.072,Z 617.884,A -85,B 0,C 180,E1 24987.545,E2 24987.545} C_VEL
LIN {X 0,Y 292.722,Z 582.007,A -85,B 0,C 180,E1 24998.822,E2 24998.822} C_VEL
LIN {X 0,Y 285.933,Z 561.672,A -85,B 0,C 180,E1 25009.39,E2 25009.39} C_VEL
LIN {X 0,Y 284.152,Z 553.373,A -85,B 0,C 180,E1 25020.856,E2 25020.856} C_VEL
LIN {X 0,Y 287.701,Z 565.615,A -85,B 0,C 180,E1 25032.801,E2 25032.801} C_VEL
LIN {X 0,Y 295.97,Z 589.145,A -85,B 0,C 180,E1 25043.212,E2 25043.212} C_VEL
LIN {X 0,Y 302.606,Z 623.063,A -85,B 0,C 180,E1 25052.506,E2 25052.506} C_VEL
LIN {X 0,Y 301.586,Z 634.294,A -85,B 0,C 180,E1 25054.574,E2 25054.574} C_VEL
LIN {X 0,Y 274.762,Z 685.107,A -85,B 0,C 180,E1 25061.236,E2 25061.236} C_VEL
LIN {X 0,Y 247.034,Z 726.384,A -85,B 0,C 180,E1 25071.57,E2 25071.57} C_VEL
LIN {X 0,Y 227.312,Z 753.98,A -85,B 0,C 180,E1 25085.357,E2 25085.357} C_VEL
LIN {X 0,Y 220.022,Z 767.364,A -85,B 0,C 180,E1 25100.078,E2 25100.078} C_VEL
LIN {X 0,Y 219.677,Z 769.724,A -85,B 0,C 180,E1 25111.978,E2 25111.978} C_VEL
LIN {X 0,Y 222.574,Z 761.802,A -85,B 0,C 180,E1 25127.854,E2 25127.854} C_VEL
LIN {X 0,Y 237.249,Z 739.914,A -85,B 0,C 180,E1 25142.909,E2 25142.909} C_VEL
LIN {X 0,Y 262.815,Z 703.663,A -85,B 0,C 180,E1 25154.979,E2 25154.979} C_VEL
LIN {X 0,Y 290.767,Z 656.58,A -85,B 0,C 180,E1 25163.013,E2 25163.013} C_VEL
LIN {X 0,Y 302.975,Z 628.263,A -85,B 0,C 180,E1 25166.292,E2 25166.292} C_VEL
LIN {X 0,Y 297.418,Z 593.559,A -85,B 0,C 180,E1 25175.233,E2 25175.233} C_VEL
LIN {X 0,Y 288.991,Z 568.986,A -85,B 0,C 180,E1 25185.265,E2 25185.265} C_VEL
LIN {X 0,Y 284.659,Z 558.333,A -85,B 0,C 180,E1 25193.405,E2 25193.405} C_VEL
LIN {X 0,Y 284.073,Z 553.717,A -85,B 0,C 180,E1 25201.63,E2 25201.63} C_VEL
LIN {X 0,Y 287.463,Z 566.393,A -85,B 0,C 180,E1 25213.646,E2 25213.646} C_VEL
LIN {X 0,Y 295.001,Z 589.676,A -85,B 0,C 180,E1 25224.034,E2 25224.034} C_VEL
LIN {X 0,Y 311.528,Z 640.584,A -85,B 0,C 180,E1 25240.096,E2 25240.096} C_VEL
LIN {X 0,Y 329.218,Z 663.012,A -85,B 0,C 180,E1 25248.283,E2 25248.283} C_VEL
LIN {X 0,Y 335.317,Z 681.699,A -85,B 0,C 180,E1 25253.401,E2 25253.401} C_VEL
LIN {X 0,Y 357.702,Z 706.139,A -85,B 0,C 180,E1 25262.483,E2 25262.483} C_VEL
LIN {X 0,Y 374.187,Z 722.979,A -85,B 0,C 180,E1 25270.89,E2 25270.89} C_VEL
LIN {X 0,Y 384.705,Z 733.072,A -85,B 0,C 180,E1 25278.633,E2 25278.633} C_VEL
LIN {X 0,Y 390.223,Z 738.081,A -85,B 0,C 180,E1 25286.658,E2 25286.658} C_VEL
LIN {X 0,Y 390.001,Z 738.122,A -85,B 0,C 180,E1 25293.344,E2 25293.344} C_VEL
LIN {X 0,Y 384.704,Z 733.086,A -85,B 0,C 180,E1 25301.367,E2 25301.367} C_VEL
LIN {X 0,Y 374.179,Z 722.904,A -85,B 0,C 180,E1 25309.128,E2 25309.128} C_VEL
LIN {X 0,Y 357.561,Z 706.138,A -85,B 0,C 180,E1 25317.532,E2 25317.532} C_VEL
LIN {X 0,Y 334.16,Z 680.903,A -85,B 0,C 180,E1 25326.944,E2 25326.944} C_VEL
LIN {X 0,Y 298.607,Z 632.106,A -85,B 0,C 180,E1 25345.065,E2 25345.065} C_VEL
LIN {X 0,Y 289.137,Z 589.737,A -85,B 0,C 180,E1 25358.789,E2 25358.789} C_VEL
LIN {X 0,Y 283.293,Z 569.561,A -85,B 0,C 180,E1 25369.29,E2 25369.29} C_VEL
LIN {X 0,Y 281.619,Z 561.176,A -85,B 0,C 180,E1 25378.549,E2 25378.549} C_VEL
LIN {X 0,Y 283.863,Z 570.695,A -85,B 0,C 180,E1 25390.875,E2 25390.875} C_VEL
LIN {X 0,Y 290.78,Z 591.73,A -85,B 0,C 180,E1 25401.399,E2 25401.399} C_VEL
LIN {X 0,Y 296.752,Z 624.249,A -85,B 0,C 180,E1 25411.013,E2 25411.013} C_VEL
LIN {X 0,Y 296.408,Z 635.695,A -85,B 0,C 180,E1 25413.439,E2 25413.439} C_VEL
LIN {X 0,Y 267.672,Z 687.846,A -85,B 0,C 180,E1 25420.447,E2 25420.447} C_VEL
LIN {X 0,Y 238.98,Z 728.552,A -85,B 0,C 180,E1 25431.197,E2 25431.197} C_VEL
LIN {X 0,Y 219.057,Z 755.07,A -85,B 0,C 180,E1 25445.457,E2 25445.457} C_VEL
LIN {X 0,Y 212.073,Z 767.187,A -85,B 0,C 180,E1 25459.702,E2 25459.702} C_VEL
LIN {X 0,Y 211.66,Z 769.548,A -85,B 0,C 180,E1 25472.053,E2 25472.053} C_VEL
LIN {X 0,Y 214.867,Z 761.625,A -85,B 0,C 180,E1 25488.518,E2 25488.518} C_VEL
LIN {X 0,Y 231.725,Z 738.256,A -85,B 0,C 180,E1 25504.742,E2 25504.742} C_VEL
LIN {X 0,Y 258.194,Z 701.985,A -85,B 0,C 180,E1 25516.622,E2 25516.622} C_VEL
LIN {X 0,Y 286.906,Z 654.64,A -85,B 0,C 180,E1 25524.528,E2 25524.528} C_VEL
LIN {X 0,Y 297.207,Z 631.015,A -85,B 0,C 180,E1 25527.342,E2 25527.342} C_VEL
LIN {X 0,Y 292.375,Z 597.073,A -85,B 0,C 180,E1 25536.594,E2 25536.594} C_VEL
LIN {X 0,Y 284.917,Z 573.356,A -85,B 0,C 180,E1 25547.255,E2 25547.255} C_VEL
LIN {X 0,Y 281.573,Z 561.705,A -85,B 0,C 180,E1 25558.364,E2 25558.364} C_VEL
LIN {X 0,Y 281.482,Z 564.987,A -85,B 0,C 180,E1 25565.68,E2 25565.68} C_VEL
LIN {X 0,Y 286.32,Z 579.823,A -85,B 0,C 180,E1 25576.85,E2 25576.85} C_VEL
LIN {X 0,Y 292.768,Z 606.944,A -85,B 0,C 180,E1 25587.095,E2 25587.095} C_VEL
LIN {X 0,Y 309.139,Z 651.098,A -85,B 0,C 180,E1 25601.917,E2 25601.917} C_VEL
LIN {X 0,Y 335.317,Z 681.699,A -85,B 0,C 180,E1 25613.401,E2 25613.401} C_VEL
LIN {X 0,Y 341.022,Z 699.384,A -85,B 0,C 180,E1 25618.549,E2 25618.549} C_VEL
LIN {X 0,Y 360.154,Z 719.377,A -85,B 0,C 180,E1 25627.126,E2 25627.126} C_VEL
LIN {X 0,Y 372.412,Z 731.841,A -85,B 0,C 180,E1 25634.652,E2 25634.652} C_VEL
LIN {X 0,Y 379.864,Z 739.317,A -85,B 0,C 180,E1 25641.968,E2 25641.968} C_VEL
LIN {X 0,Y 383.352,Z 741.772,A -85,B 0,C 180,E1 25648.867,E2 25648.867} C_VEL
LIN {X 0,Y 381.581,Z 740.541,A -85,B 0,C 180,E1 25655.702,E2 25655.702} C_VEL
LIN {X 0,Y 374.376,Z 733.49,A -85,B 0,C 180,E1 25663.982,E2 25663.982} C_VEL
LIN {X 0,Y 360.879,Z 720.325,A -85,B 0,C 180,E1 25672.424,E2 25672.424} C_VEL
LIN {X 0,Y 341.888,Z 700.657,A -85,B 0,C 180,E1 25681.007,E2 25681.007} C_VEL
LIN {X 0,Y 312.073,Z 668.341,A -85,B 0,C 180,E1 25693.412,E2 25693.412} C_VEL
LIN {X 0,Y 289.113,Z 623.371,A -85,B 0,C 180,E1 25710.2,E2 25710.2} C_VEL
LIN {X 0,Y 284.32,Z 593.155,A -85,B 0,C 180,E1 25720.513,E2 25720.513} C_VEL
LIN {X 0,Y 279.858,Z 575.224,A -85,B 0,C 180,E1 25730.734,E2 25730.734} C_VEL
LIN {X 0,Y 279.014,Z 568.909,A -85,B 0,C 180,E1 25738.535,E2 25738.535} C_VEL
LIN {X 0,Y 280.942,Z 578.386,A -85,B 0,C 180,E1 25750.99,E2 25750.99} C_VEL
LIN {X 0,Y 286.889,Z 599.458,A -85,B 0,C 180,E1 25761.419,E2 25761.419} C_VEL
LIN {X 0,Y 291.403,Z 631.497,A -85,B 0,C 180,E1 25771.001,E2 25771.001} C_VEL
LIN {X 0,Y 289.274,Z 641.031,A -85,B 0,C 180,E1 25772.672,E2 25772.672} C_VEL
LIN {X 0,Y 259.735,Z 691.661,A -85,B 0,C 180,E1 25779.879,E2 25779.879} C_VEL
LIN {X 0,Y 230.954,Z 730.581,A -85,B 0,C 180,E1 25790.802,E2 25790.802} C_VEL
LIN {X 0,Y 209.983,Z 757.346,A -85,B 0,C 180,E1 25806.596,E2 25806.596} C_VEL
LIN {X 0,Y 203.481,Z 768.581,A -85,B 0,C 180,E1 25823.581,E2 25823.581} C_VEL
LIN {X 0,Y 203.557,Z 768.583,A -85,B 0,C 180,E1 25836.416,E2 25836.416} C_VEL
LIN {X 0,Y 210.001,Z 757.347,A -85,B 0,C 180,E1 25853.401,E2 25853.401} C_VEL
LIN {X 0,Y 231.034,Z 730.584,A -85,B 0,C 180,E1 25869.181,E2 25869.181} C_VEL
LIN {X 0,Y 259.845,Z 691.445,A -85,B 0,C 180,E1 25880.175,E2 25880.175} C_VEL
LIN {X 0,Y 289.269,Z 641.034,A -85,B 0,C 180,E1 25887.329,E2 25887.329} C_VEL
LIN {X 0,Y 291.34,Z 629.947,A -85,B 0,C 180,E1 25889.382,E2 25889.382} C_VEL
LIN {X 0,Y 287.064,Z 599.059,A -85,B 0,C 180,E1 25898.595,E2 25898.595} C_VEL
LIN {X 0,Y 280.95,Z 578.366,A -85,B 0,C 180,E1 25909.011,E2 25909.011} C_VEL
LIN {X 0,Y 278.975,Z 569.419,A -85,B 0,C 180,E1 25918.348,E2 25918.348} C_VEL
LIN {X 0,Y 279.334,Z 573.889,A -85,B 0,C 180,E1 25927.71,E2 25927.71} C_VEL
LIN {X 0,Y 283.964,Z 591.518,A -85,B 0,C 180,E1 25938.785,E2 25938.785} C_VEL
LIN {X 0,Y 288.572,Z 618.539,A -85,B 0,C 180,E1 25948.346,E2 25948.346} C_VEL
LIN {X 0,Y 306.793,Z 661.278,A -85,B 0,C 180,E1 25963.847,E2 25963.847} C_VEL
LIN {X 0,Y 337.294,Z 695.426,A -85,B 0,C 180,E1 25977.079,E2 25977.079} C_VEL
LIN {X 0,Y 341.022,Z 699.384,A -85,B 0,C 180,E1 25978.549,E2 25978.549} C_VEL
LIN {X 0,Y 345.591,Z 715.43,A -85,B 0,C 180,E1 25983.805,E2 25983.805} C_VEL
LIN {X 0,Y 360.446,Z 730.4,A -85,B 0,C 180,E1 25991.606,E2 25991.606} C_VEL
LIN {X 0,Y 370.597,Z 740.095,A -85,B 0,C 180,E1 25999.389,E2 25999.389} C_VEL
LIN {X 0,Y 375.403,Z 744.414,A -85,B 0,C 180,E1 26006.526,E2 26006.526} C_VEL
LIN {X 0,Y 375.223,Z 744.431,A -85,B 0,C 180,E1 26013.476,E2 26013.476} C_VEL
LIN {X 0,Y 369.45,Z 738.828,A -85,B 0,C 180,E1 26021.843,E2 26021.843} C_VEL
LIN {X 0,Y 356.829,Z 726.892,A -85,B 0,C 180,E1 26030.491,E2 26030.491} C_VEL
LIN {X 0,Y 340.359,Z 710.018,A -85,B 0,C 180,E1 26038.505,E2 26038.505} C_VEL
LIN {X 0,Y 312.325,Z 680.53,A -85,B 0,C 180,E1 26050.273,E2 26050.273} C_VEL
LIN {X 0,Y 284.815,Z 634.278,A -85,B 0,C 180,E1 26068.816,E2 26068.816} C_VEL
LIN {X 0,Y 280.301,Z 599.864,A -85,B 0,C 180,E1 26080.889,E2 26080.889} C_VEL
LIN {X 0,Y 276.785,Z 582.953,A -85,B 0,C 180,E1 26090.63,E2 26090.63} C_VEL
LIN {X 0,Y 276.102,Z 576.52,A -85,B 0,C 180,E1 26098.52,E2 26098.52} C_VEL
LIN {X 0,Y 277.887,Z 586.114,A -85,B 0,C 180,E1 26111.112,E2 26111.112} C_VEL
LIN {X 0,Y 282.938,Z 607.448,A -85,B 0,C 180,E1 26121.567,E2 26121.567} C_VEL
LIN {X 0,Y 285.875,Z 638.003,A -85,B 0,C 180,E1 26130.824,E2 26130.824} C_VEL
LIN {X 0,Y 256.034,Z 689.51,A -85,B 0,C 180,E1 26138.079,E2 26138.079} C_VEL
LIN {X 0,Y 225.592,Z 729.358,A -85,B 0,C 180,E1 26149.048,E2 26149.048} C_VEL
LIN {X 0,Y 203.794,Z 755.438,A -85,B 0,C 180,E1 26164.161,E2 26164.161} C_VEL
LIN {X 0,Y 196.218,Z 766.835,A -85,B 0,C 180,E1 26178.859,E2 26178.859} C_VEL
LIN {X 0,Y 195.647,Z 769.198,A -85,B 0,C 180,E1 26192.221,E2 26192.221} C_VEL
LIN {X 0,Y 199.542,Z 761.27,A -85,B 0,C 180,E1 26209.998,E2 26209.998} C_VEL
LIN {X 0,Y 218.797,Z 737.585,A -85,B 0,C 180,E1 26227.334,E2 26227.334} C_VEL
LIN {X 0,Y 248.48,Z 700.127,A -85,B 0,C 180,E1 26239.719,E2 26239.719} C_VEL
LIN {X 0,Y 279.596,Z 651.211,A -85,B 0,C 180,E1 26247.61,E2 26247.61} C_VEL
LIN {X 0,Y 285.865,Z 638.02,A -85,B 0,C 180,E1 26249.174,E2 26249.174} C_VEL
LIN {X 0,Y 283.111,Z 606.967,A -85,B 0,C 180,E1 26258.487,E2 26258.487} C_VEL
LIN {X 0,Y 277.898,Z 586.087,A -85,B 0,C 180,E1 26268.888,E2 26268.888} C_VEL
LIN {X 0,Y 276.06,Z 577.011,A -85,B 0,C 180,E1 26278.331,E2 26278.331} C_VEL
LIN {X 0,Y 276.293,Z 581.508,A -85,B 0,C 180,E1 26287.796,E2 26287.796} C_VEL
LIN {X 0,Y 280.316,Z 599.864,A -85,B 0,C 180,E1 26299.12,E2 26299.12} C_VEL
LIN {X 0,Y 284.245,Z 630.457,A -85,B 0,C 180,E1 26309.921,E2 26309.921} C_VEL
LIN {X 0,Y 307.755,Z 674.69,A -85,B 0,C 180,E1 26327.412,E2 26327.412} C_VEL
LIN {X 0,Y 337.018,Z 706.277,A -85,B 0,C 180,E1 26340.029,E2 26340.029} C_VEL
LIN {X 0,Y 345.591,Z 715.43,A -85,B 0,C 180,E1 26343.805,E2 26343.805} C_VEL
LIN {X 0,Y 348.812,Z 729.03,A -85,B 0,C 180,E1 26349.228,E2 26349.228} C_VEL
LIN {X 0,Y 361.56,Z 741.292,A -85,B 0,C 180,E1 26357.896,E2 26357.896} C_VEL
LIN {X 0,Y 367.79,Z 747.04,A -85,B 0,C 180,E1 26366.454,E2 26366.454} C_VEL
LIN {X 0,Y 367.629,Z 747.046,A -85,B 0,C 180,E1 26373.548,E2 26373.548} C_VEL
LIN {X 0,Y 361.56,Z 741.245,A -85,B 0,C 180,E1 26382.104,E2 26382.104} C_VEL
LIN {X 0,Y 350.353,Z 730.7,A -85,B 0,C 180,E1 26389.835,E2 26389.835} C_VEL
LIN {X 0,Y 334.109,Z 714.188,A -85,B 0,C 180,E1 26397.853,E2 26397.853} C_VEL
LIN {X 0,Y 306.147,Z 685.404,A -85,B 0,C 180,E1 26409.944,E2 26409.944} C_VEL
LIN {X 0,Y 279.356,Z 640.143,A -85,B 0,C 180,E1 26429.047,E2 26429.047} C_VEL
LIN {X 0,Y 276.109,Z 606.917,A -85,B 0,C 180,E1 26441.056,E2 26441.056} C_VEL
LIN {X 0,Y 273.204,Z 588.869,A -85,B 0,C 180,E1 26452.116,E2 26452.116} C_VEL
LIN {X 0,Y 273.053,Z 584.09,A -85,B 0,C 180,E1 26458.503,E2 26458.503} C_VEL
LIN {X 0,Y 274.154,Z 592.352,A -85,B 0,C 180,E1 26470.171,E2 26470.171} C_VEL
LIN {X 0,Y 278.283,Z 612.993,A -85,B 0,C 180,E1 26480.856,E2 26480.856} C_VEL
LIN {X 0,Y 280.048,Z 642.261,A -85,B 0,C 180,E1 26490.056,E2 26490.056} C_VEL
LIN {X 0,Y 248.553,Z 692.77,A -85,B 0,C 180,E1 26497.316,E2 26497.316} C_VEL
LIN {X 0,Y 217.614,Z 731.252,A -85,B 0,C 180,E1 26508.545,E2 26508.545} C_VEL
LIN {X 0,Y 195.122,Z 756.99,A -85,B 0,C 180,E1 26524.693,E2 26524.693} C_VEL
LIN {X 0,Y 187.502,Z 768.229,A -85,B 0,C 180,E1 26543.032,E2 26543.032} C_VEL
LIN {X 0,Y 187.568,Z 768.231,A -85,B 0,C 180,E1 26556.965,E2 26556.965} C_VEL
LIN {X 0,Y 195.138,Z 756.991,A -85,B 0,C 180,E1 26575.304,E2 26575.304} C_VEL
LIN {X 0,Y 217.683,Z 731.254,A -85,B 0,C 180,E1 26591.438,E2 26591.438} C_VEL
LIN {X 0,Y 248.16,Z 693.243,A -85,B 0,C 180,E1 26602.6,E2 26602.6} C_VEL
LIN {X 0,Y 279.235,Z 643.802,A -85,B 0,C 180,E1 26609.788,E2 26609.788} C_VEL
LIN {X 0,Y 279.253,Z 618.268,A -85,B 0,C 180,E1 26617.124,E2 26617.124} C_VEL
LIN {X 0,Y 275.034,Z 596.221,A -85,B 0,C 180,E1 26627.155,E2 26627.155} C_VEL
LIN {X 0,Y 273.012,Z 584.583,A -85,B 0,C 180,E1 26638.312,E2 26638.312} C_VEL
LIN {X 0,Y 272.817,Z 587.835,A -85,B 0,C 180,E1 26646.29,E2 26646.29} C_VEL
LIN {X 0,Y 275.708,Z 603.813,A -85,B 0,C 180,E1 26657.519,E2 26657.519} C_VEL
LIN {X 0,Y 278.212,Z 630.17,A -85,B 0,C 180,E1 26667.51,E2 26667.51} C_VEL
LIN {X 0,Y 295.424,Z 672.591,A -85,B 0,C 180,E1 26684.476,E2 26684.476} C_VEL
LIN {X 0,Y 325.655,Z 705.231,A -85,B 0,C 180,E1 26698.457,E2 26698.457} C_VEL
LIN {X 0,Y 345.617,Z 725.709,A -85,B 0,C 180,E1 26707.458,E2 26707.458} C_VEL
LIN {X 0,Y 348.812,Z 729.03,A -85,B 0,C 180,E1 26709.228,E2 26709.228} C_VEL
LIN {X 0,Y 349.769,Z 740.05,A -85,B 0,C 180,E1 26714.787,E2 26714.787} C_VEL
LIN {X 0,Y 356.817,Z 746.965,A -85,B 0,C 180,E1 26721.446,E2 26721.446} C_VEL
LIN {X 0,Y 360.779,Z 749.895,A -85,B 0,C 180,E1 26728.796,E2 26728.796} C_VEL
LIN {X 0,Y 358.388,Z 748.294,A -85,B 0,C 180,E1 26736.491,E2 26736.491} C_VEL
LIN {X 0,Y 351.443,Z 741.44,A -85,B 0,C 180,E1 26744.057,E2 26744.057} C_VEL
LIN {X 0,Y 337.879,Z 728.316,A -85,B 0,C 180,E1 26752.427,E2 26752.427} C_VEL
LIN {X 0,Y 316.513,Z 706.993,A -85,B 0,C 180,E1 26762.074,E2 26762.074} C_VEL
LIN {X 0,Y 285.881,Z 674.057,A -85,B 0,C 180,E1 26777.151,E2 26777.151} C_VEL
LIN {X 0,Y 272.6,Z 631.159,A -85,B 0,C 180,E1 26794.604,E2 26794.604} C_VEL
LIN {X 0,Y 271.088,Z 607.016,A -85,B 0,C 180,E1 26804.556,E2 26804.556} C_VEL
LIN {X 0,Y 269.443,Z 595.049,A -85,B 0,C 180,E1 26813.631,E2 26813.631} C_VEL
LIN {X 0,Y 269.714,Z 592.003,A -85,B 0,C 180,E1 26821.708,E2 26821.708} C_VEL
LIN {X 0,Y 271.713,Z 605.288,A -85,B 0,C 180,E1 26833.826,E2 26833.826} C_VEL
LIN {X 0,Y 274.451,Z 628.995,A -85,B 0,C 180,E1 26843.955,E2 26843.955} C_VEL
LIN {X 0,Y 273.662,Z 646.638,A -85,B 0,C 180,E1 26849.07,E2 26849.07} C_VEL
LIN {X 0,Y 242.076,Z 694.753,A -85,B 0,C 180,E1 26856.239,E2 26856.239} C_VEL
LIN {X 0,Y 209.663,Z 733.128,A -85,B 0,C 180,E1 26868.006,E2 26868.006} C_VEL
LIN {X 0,Y 186.845,Z 757.841,A -85,B 0,C 180,E1 26884.779,E2 26884.779} C_VEL
LIN {X 0,Y 179.517,Z 768.053,A -85,B 0,C 180,E1 26902.72,E2 26902.72} C_VEL
LIN {X 0,Y 179.578,Z 768.055,A -85,B 0,C 180,E1 26917.277,E2 26917.277} C_VEL
LIN {X 0,Y 187.812,Z 756.813,A -85,B 0,C 180,E1 26936.365,E2 26936.365} C_VEL
LIN {X 0,Y 211.599,Z 731.075,A -85,B 0,C 180,E1 26952.91,E2 26952.91} C_VEL
LIN {X 0,Y 243.328,Z 693.066,A -85,B 0,C 180,E1 26964.115,E2 26964.115} C_VEL
LIN {X 0,Y 274.591,Z 643.812,A -85,B 0,C 180,E1 26971.431,E2 26971.431} C_VEL
LIN {X 0,Y 273.694,Z 616.68,A -85,B 0,C 180,E1 26980.472,E2 26980.472} C_VEL
LIN {X 0,Y 270.158,Z 597.281,A -85,B 0,C 180,E1 26991.832,E2 26991.832} C_VEL
LIN {X 0,Y 269.697,Z 591.663,A -85,B 0,C 180,E1 27001.515,E2 27001.515} C_VEL
LIN {X 0,Y 270.616,Z 603.776,A -85,B 0,C 180,E1 27013.472,E2 27013.472} C_VEL
LIN {X 0,Y 272.753,Z 626.79,A -85,B 0,C 180,E1 27023.99,E2 27023.99} C_VEL
LIN {X 0,Y 282.797,Z 668.982,A -85,B 0,C 180,E1 27040.587,E2 27040.587} C_VEL
LIN {X 0,Y 313.353,Z 703.36,A -85,B 0,C 180,E1 27056.396,E2 27056.396} C_VEL
LIN {X 0,Y 337.134,Z 727.323,A -85,B 0,C 180,E1 27067.105,E2 27067.105} C_VEL
LIN {X 0,Y 349.769,Z 740.05,A -85,B 0,C 180,E1 27074.787,E2 27074.787} C_VEL
LIN {X 0,Y 348.297,Z 748.211,A -85,B 0,C 180,E1 27080.498,E2 27080.498} C_VEL
LIN {X 0,Y 353.058,Z 752.031,A -85,B 0,C 180,E1 27088.77,E2 27088.77} C_VEL
LIN {X 0,Y 350.864,Z 750.544,A -85,B 0,C 180,E1 27096.203,E2 27096.203} C_VEL
LIN {X 0,Y 343.662,Z 743.586,A -85,B 0,C 180,E1 27104.046,E2 27104.046} C_VEL
LIN {X 0,Y 329.83,Z 730.194,A -85,B 0,C 180,E1 27112.487,E2 27112.487} C_VEL
LIN {X 0,Y 307.598,Z 708.593,A -85,B 0,C 180,E1 27122.657,E2 27122.657} C_VEL
LIN {X 0,Y 276.819,Z 675.001,A -85,B 0,C 180,E1 27139,E2 27139} C_VEL
LIN {X 0,Y 267.505,Z 632.09,A -85,B 0,C 180,E1 27156.757,E2 27156.757} C_VEL
LIN {X 0,Y 266.6,Z 610.192,A -85,B 0,C 180,E1 27166.942,E2 27166.942} C_VEL
LIN {X 0,Y 266.283,Z 598.9,A -85,B 0,C 180,E1 27178.465,E2 27178.465} C_VEL
LIN {X 0,Y 266.741,Z 606.018,A -85,B 0,C 180,E1 27189.363,E2 27189.363} C_VEL
LIN {X 0,Y 268.925,Z 624.661,A -85,B 0,C 180,E1 27199.675,E2 27199.675} C_VEL
LIN {X 0,Y 268.23,Z 649.373,A -85,B 0,C 180,E1 27207.868,E2 27207.868} C_VEL
LIN {X 0,Y 234.747,Z 697.948,A -85,B 0,C 180,E1 27215.354,E2 27215.354} C_VEL
LIN {X 0,Y 201.721,Z 735.004,A -85,B 0,C 180,E1 27227.421,E2 27227.421} C_VEL
LIN {X 0,Y 178.568,Z 758.691,A -85,B 0,C 180,E1 27244.873,E2 27244.873} C_VEL
LIN {X 0,Y 171.537,Z 767.878,A -85,B 0,C 180,E1 27262.379,E2 27262.379} C_VEL
LIN {X 0,Y 171.623,Z 767.88,A -85,B 0,C 180,E1 27277.616,E2 27277.616} C_VEL
LIN {X 0,Y 180.99,Z 756.162,A -85,B 0,C 180,E1 27298.029,E2 27298.029} C_VEL
LIN {X 0,Y 206.893,Z 729.663,A -85,B 0,C 180,E1 27315.018,E2 27315.018} C_VEL
LIN {X 0,Y 241.295,Z 689.515,A -85,B 0,C 180,E1 27326.38,E2 27326.38} C_VEL
LIN {X 0,Y 269.104,Z 646.838,A -85,B 0,C 180,E1 27332.596,E2 27332.596} C_VEL
LIN {X 0,Y 268.899,Z 620.901,A -85,B 0,C 180,E1 27341.819,E2 27341.819} C_VEL
LIN {X 0,Y 266.593,Z 604.754,A -85,B 0,C 180,E1 27351.722,E2 27351.722} C_VEL
LIN {X 0,Y 266.225,Z 599.024,A -85,B 0,C 180,E1 27361.535,E2 27361.535} C_VEL
LIN {X 0,Y 266.656,Z 611.674,A -85,B 0,C 180,E1 27373.893,E2 27373.893} C_VEL
LIN {X 0,Y 267.572,Z 633.766,A -85,B 0,C 180,E1 27383.912,E2 27383.912} C_VEL
LIN {X 0,Y 277.042,Z 674.708,A -85,B 0,C 180,E1 27400.96,E2 27400.96} C_VEL
LIN {X 0,Y 306.92,Z 707.522,A -85,B 0,C 180,E1 27416.891,E2 27416.891} C_VEL
LIN {X 0,Y 329.976,Z 730.149,A -85,B 0,C 180,E1 27427.513,E2 27427.513} C_VEL
LIN {X 0,Y 343.623,Z 743.61,A -85,B 0,C 180,E1 27435.953,E2 27435.953} C_VEL
LIN {X 0,Y 348.297,Z 748.211,A -85,B 0,C 180,E1 27440.498,E2 27440.498} C_VEL
LIN {X 0,Y 344.412,Z 753.325,A -85,B 0,C 180,E1 27446.293,E2 27446.293} C_VEL
LIN {X 0,Y 344.283,Z 753.302,A -85,B 0,C 180,E1 27453.788,E2 27453.788} C_VEL
LIN {X 0,Y 338.676,Z 748.077,A -85,B 0,C 180,E1 27461.625,E2 27461.625} C_VEL
LIN {X 0,Y 325.523,Z 735.679,A -85,B 0,C 180,E1 27470.451,E2 27470.451} C_VEL
LIN {X 0,Y 304.572,Z 715.755,A -85,B 0,C 180,E1 27480.53,E2 27480.53} C_VEL
LIN {X 0,Y 275.343,Z 686.462,A -85,B 0,C 180,E1 27495.5,E2 27495.5} C_VEL
LIN {X 0,Y 261.799,Z 645.635,A -85,B 0,C 180,E1 27514.347,E2 27514.347} C_VEL
LIN {X 0,Y 262.507,Z 622.236,A -85,B 0,C 180,E1 27524.168,E2 27524.168} C_VEL
LIN {X 0,Y 262.101,Z 609.574,A -85,B 0,C 180,E1 27533.452,E2 27533.452} C_VEL
LIN {X 0,Y 262.582,Z 606.581,A -85,B 0,C 180,E1 27541.755,E2 27541.755} C_VEL
LIN {X 0,Y 263.462,Z 619.089,A -85,B 0,C 180,E1 27553.419,E2 27553.419} C_VEL
LIN {X 0,Y 264.052,Z 641.5,A -85,B 0,C 180,E1 27563.375,E2 27563.375} C_VEL
LIN {X 0,Y 262.157,Z 653.012,A -85,B 0,C 180,E1 27566.746,E2 27566.746} C_VEL
LIN {X 0,Y 227.583,Z 700.811,A -85,B 0,C 180,E1 27574.391,E2 27574.391} C_VEL
LIN {X 0,Y 193.806,Z 736.869,A -85,B 0,C 180,E1 27586.79,E2 27586.79} C_VEL
LIN {X 0,Y 169.39,Z 760.56,A -85,B 0,C 180,E1 27606.242,E2 27606.242} C_VEL
LIN {X 0,Y 163.273,Z 768.49,A -85,B 0,C 180,E1 27627.338,E2 27627.338} C_VEL
LIN {X 0,Y 164.881,Z 765.702,A -85,B 0,C 180,E1 27644.315,E2 27644.315} C_VEL
LIN {X 0,Y 179.781,Z 750.105,A -85,B 0,C 180,E1 27664.706,E2 27664.706} C_VEL
LIN {X 0,Y 211.112,Z 719.213,A -85,B 0,C 180,E1 27680.552,E2 27680.552} C_VEL
LIN {X 0,Y 246.785,Z 676.232,A -85,B 0,C 180,E1 27690.252,E2 27690.252} C_VEL
LIN {X 0,Y 263.672,Z 649.577,A -85,B 0,C 180,E1 27693.911,E2 27693.911} C_VEL
LIN {X 0,Y 264.063,Z 625.48,A -85,B 0,C 180,E1 27703.007,E2 27703.007} C_VEL
LIN {X 0,Y 262.518,Z 610.298,A -85,B 0,C 180,E1 27713.263,E2 27713.263} C_VEL
LIN {X 0,Y 262.551,Z 606.266,A -85,B 0,C 180,E1 27721.557,E2 27721.557} C_VEL
LIN {X 0,Y 262.417,Z 617.873,A -85,B 0,C 180,E1 27733.27,E2 27733.27} C_VEL
LIN {X 0,Y 262.319,Z 639.033,A -85,B 0,C 180,E1 27743.282,E2 27743.282} C_VEL
LIN {X 0,Y 270.451,Z 679.186,A -85,B 0,C 180,E1 27760.801,E2 27760.801} C_VEL
LIN {X 0,Y 300.026,Z 711.149,A -85,B 0,C 180,E1 27777.234,E2 27777.234} C_VEL
LIN {X 0,Y 323.533,Z 733.433,A -85,B 0,C 180,E1 27788.366,E2 27788.366} C_VEL
LIN {X 0,Y 337.295,Z 746.804,A -85,B 0,C 180,E1 27797.192,E2 27797.192} C_VEL
LIN {X 0,Y 344.412,Z 753.325,A -85,B 0,C 180,E1 27806.293,E2 27806.293} C_VEL
LIN {X 0,Y 336.887,Z 755.174,A -85,B 0,C 180,E1 27812.146,E2 27812.146} C_VEL
LIN {X 0,Y 331.547,Z 750.394,A -85,B 0,C 180,E1 27820.733,E2 27820.733} C_VEL
LIN {X 0,Y 320.636,Z 740.135,A -85,B 0,C 180,E1 27828.638,E2 27828.638} C_VEL
LIN {X 0,Y 301.308,Z 722.346,A -85,B 0,C 180,E1 27838.395,E2 27838.395} C_VEL
LIN {X 0,Y 272.974,Z 695.749,A -85,B 0,C 180,E1 27852.712,E2 27852.712} C_VEL
LIN {X 0,Y 256.001,Z 656.015,A -85,B 0,C 180,E1 27872.772,E2 27872.772} C_VEL
LIN {X 0,Y 257.933,Z 629.878,A -85,B 0,C 180,E1 27883.88,E2 27883.88} C_VEL
LIN {X 0,Y 258.205,Z 616.739,A -85,B 0,C 180,E1 27893.353,E2 27893.353} C_VEL
LIN {X 0,Y 258.705,Z 613.701,A -85,B 0,C 180,E1 27901.781,E2 27901.781} C_VEL
LIN {X 0,Y 258.945,Z 625.079,A -85,B 0,C 180,E1 27912.797,E2 27912.797} C_VEL
LIN {X 0,Y 258.703,Z 647.333,A -85,B 0,C 180,E1 27922.962,E2 27922.962} C_VEL
LIN {X 0,Y 256.06,Z 656.791,A -85,B 0,C 180,E1 27925.577,E2 27925.577} C_VEL
LIN {X 0,Y 219.335,Z 704.805,A -85,B 0,C 180,E1 27933.675,E2 27933.675} C_VEL
LIN {X 0,Y 184.452,Z 739.79,A -85,B 0,C 180,E1 27946.859,E2 27946.859} C_VEL
LIN {X 0,Y 161.966,Z 760.382,A -85,B 0,C 180,E1 27965.081,E2 27965.081} C_VEL
LIN {X 0,Y 155.284,Z 768.315,A -85,B 0,C 180,E1 27987.201,E2 27987.201} C_VEL
LIN {X 0,Y 157.596,Z 764.819,A -85,B 0,C 180,E1 28006.779,E2 28006.779} C_VEL
LIN {X 0,Y 176.43,Z 746.892,A -85,B 0,C 180,E1 28028.547,E2 28028.547} C_VEL
LIN {X 0,Y 209.797,Z 715.046,A -85,B 0,C 180,E1 28043.528,E2 28043.528} C_VEL
LIN {X 0,Y 247.23,Z 669.838,A -85,B 0,C 180,E1 28052.8,E2 28052.8} C_VEL
LIN {X 0,Y 258.187,Z 652.653,A -85,B 0,C 180,E1 28055.123,E2 28055.123} C_VEL
LIN {X 0,Y 259.241,Z 628.992,A -85,B 0,C 180,E1 28064.841,E2 28064.841} C_VEL
LIN {X 0,Y 258.481,Z 616.131,A -85,B 0,C 180,E1 28074.848,E2 28074.848} C_VEL
LIN {X 0,Y 258.671,Z 613.391,A -85,B 0,C 180,E1 28081.58,E2 28081.58} C_VEL
LIN {X 0,Y 257.966,Z 624.334,A -85,B 0,C 180,E1 28092.926,E2 28092.926} C_VEL
LIN {X 0,Y 256.911,Z 645.412,A -85,B 0,C 180,E1 28103.066,E2 28103.066} C_VEL
LIN {X 0,Y 264.424,Z 684.487,A -85,B 0,C 180,E1 28121.157,E2 28121.157} C_VEL
LIN {X 0,Y 294.2,Z 715.691,A -85,B 0,C 180,E1 28138.144,E2 28138.144} C_VEL
LIN {X 0,Y 316.501,Z 735.999,A -85,B 0,C 180,E1 28148.961,E2 28148.961} C_VEL
LIN {X 0,Y 329.012,Z 748.008,A -85,B 0,C 180,E1 28156.97,E2 28156.97} C_VEL
LIN {X 0,Y 334.747,Z 753.708,A -85,B 0,C 180,E1 28163.497,E2 28163.497} C_VEL
LIN {X 0,Y 337.267,Z 755.355,A -85,B 0,C 180,E1 28171.288,E2 28171.288} C_VEL
LIN {X 0,Y 336.887,Z 755.174,A -85,B 0,C 180,E1 28172.146,E2 28172.146} C_VEL
LIN {X 0,Y 325.763,Z 753.886,A -85,B 0,C 180,E1 28178.014,E2 28178.014} C_VEL
LIN {X 0,Y 316.612,Z 745.081,A -85,B 0,C 180,E1 28186.13,E2 28186.13} C_VEL
LIN {X 0,Y 299.347,Z 729.673,A -85,B 0,C 180,E1 28195.506,E2 28195.506} C_VEL
LIN {X 0,Y 272.39,Z 706.123,A -85,B 0,C 180,E1 28208.913,E2 28208.913} C_VEL
LIN {X 0,Y 250.203,Z 665.972,A -85,B 0,C 180,E1 28230.992,E2 28230.992} C_VEL
LIN {X 0,Y 253.11,Z 635.689,A -85,B 0,C 180,E1 28244.458,E2 28244.458} C_VEL
LIN {X 0,Y 254.016,Z 622.51,A -85,B 0,C 180,E1 28254.963,E2 28254.963} C_VEL
LIN {X 0,Y 254.676,Z 620.731,A -85,B 0,C 180,E1 28261.809,E2 28261.809} C_VEL
LIN {X 0,Y 254.461,Z 632.47,A -85,B 0,C 180,E1 28273.026,E2 28273.026} C_VEL
LIN {X 0,Y 252.926,Z 654.348,A -85,B 0,C 180,E1 28283.061,E2 28283.061} C_VEL
LIN {X 0,Y 246.233,Z 666.067,A -85,B 0,C 180,E1 28285.036,E2 28285.036} C_VEL
LIN {X 0,Y 209.087,Z 710.879,A -85,B 0,C 180,E1 28293.479,E2 28293.479} C_VEL
LIN {X 0,Y 174.02,Z 743.643,A -85,B 0,C 180,E1 28307.517,E2 28307.517} C_VEL
LIN {X 0,Y 151.177,Z 763.401,A -85,B 0,C 180,E1 28329.446,E2 28329.446} C_VEL
LIN {X 0,Y 147.272,Z 768.14,A -85,B 0,C 180,E1 28347.049,E2 28347.049} C_VEL
LIN {X 0,Y 149.852,Z 764.642,A -85,B 0,C 180,E1 28367.673,E2 28367.673} C_VEL
LIN {X 0,Y 169.522,Z 747.232,A -85,B 0,C 180,E1 28389.861,E2 28389.861} C_VEL
LIN {X 0,Y 205.07,Z 714.868,A -85,B 0,C 180,E1 28405.355,E2 28405.355} C_VEL
LIN {X 0,Y 243.635,Z 669.661,A -85,B 0,C 180,E1 28414.494,E2 28414.494} C_VEL
LIN {X 0,Y 252.815,Z 655.565,A -85,B 0,C 180,E1 28416.461,E2 28416.461} C_VEL
LIN {X 0,Y 254.595,Z 633.774,A -85,B 0,C 180,E1 28426.102,E2 28426.102} C_VEL
LIN {X 0,Y 254.372,Z 622.012,A -85,B 0,C 180,E1 28436.367,E2 28436.367} C_VEL
LIN {X 0,Y 254.142,Z 621.603,A -85,B 0,C 180,E1 28443.392,E2 28443.392} C_VEL
LIN {X 0,Y 253.323,Z 633.572,A -85,B 0,C 180,E1 28454.345,E2 28454.345} C_VEL
LIN {X 0,Y 250.681,Z 656.666,A -85,B 0,C 180,E1 28464.938,E2 28464.938} C_VEL
LIN {X 0,Y 261.539,Z 693.975,A -85,B 0,C 180,E1 28484.08,E2 28484.08} C_VEL
LIN {X 0,Y 289.515,Z 721.085,A -85,B 0,C 180,E1 28499.669,E2 28499.669} C_VEL
LIN {X 0,Y 309.896,Z 738.776,A -85,B 0,C 180,E1 28509.826,E2 28509.826} C_VEL
LIN {X 0,Y 323.271,Z 751.324,A -85,B 0,C 180,E1 28519.011,E2 28519.011} C_VEL
LIN {X 0,Y 328.412,Z 755.981,A -85,B 0,C 180,E1 28526.028,E2 28526.028} C_VEL
LIN {X 0,Y 328.352,Z 755.968,A -85,B 0,C 180,E1 28533.973,E2 28533.973} C_VEL
LIN {X 0,Y 325.763,Z 753.886,A -85,B 0,C 180,E1 28538.014,E2 28538.014} C_VEL
LIN {X 0,Y 311.694,Z 748.911,A -85,B 0,C 180,E1 28543.858,E2 28543.858} C_VEL
LIN {X 0,Y 295.931,Z 735.33,A -85,B 0,C 180,E1 28553.155,E2 28553.155} C_VEL
LIN {X 0,Y 270.644,Z 714.522,A -85,B 0,C 180,E1 28565.789,E2 28565.789} C_VEL
LIN {X 0,Y 244.341,Z 674.554,A -85,B 0,C 180,E1 28589.534,E2 28589.534} C_VEL
LIN {X 0,Y 248.235,Z 641.463,A -85,B 0,C 180,E1 28605.053,E2 28605.053} C_VEL
LIN {X 0,Y 249.735,Z 629.416,A -85,B 0,C 180,E1 28614.876,E2 28614.876} C_VEL
LIN {X 0,Y 250.37,Z 627.697,A -85,B 0,C 180,E1 28621.976,E2 28621.976} C_VEL
LIN {X 0,Y 249.598,Z 639.699,A -85,B 0,C 180,E1 28633.283,E2 28633.283} C_VEL
LIN {X 0,Y 247.376,Z 659.147,A -85,B 0,C 180,E1 28642.344,E2 28642.344} C_VEL
LIN {X 0,Y 209.219,Z 706.068,A -85,B 0,C 180,E1 28650.384,E2 28650.384} C_VEL
LIN {X 0,Y 172.314,Z 739.91,A -85,B 0,C 180,E1 28663.443,E2 28663.443} C_VEL
LIN {X 0,Y 145.339,Z 761.635,A -85,B 0,C 180,E1 28685.331,E2 28685.331} C_VEL
LIN {X 0,Y 139.272,Z 767.965,A -85,B 0,C 180,E1 28706.879,E2 28706.879} C_VEL
LIN {X 0,Y 142.174,Z 764.465,A -85,B 0,C 180,E1 28728.662,E2 28728.662} C_VEL
LIN {X 0,Y 164.376,Z 746.246,A -85,B 0,C 180,E1 28752.319,E2 28752.319} C_VEL
LIN {X 0,Y 201.921,Z 713.36,A -85,B 0,C 180,E1 28767.662,E2 28767.662} C_VEL
LIN {X 0,Y 241.331,Z 668.057,A -85,B 0,C 180,E1 28776.411,E2 28776.411} C_VEL
LIN {X 0,Y 247.81,Z 657.174,A -85,B 0,C 180,E1 28778.351,E2 28778.351} C_VEL
LIN {X 0,Y 249.742,Z 638.183,A -85,B 0,C 180,E1 28787.617,E2 28787.617} C_VEL
LIN {X 0,Y 250.374,Z 627.645,A -85,B 0,C 180,E1 28798.16,E2 28798.16} C_VEL
LIN {X 0,Y 249.456,Z 630.986,A -85,B 0,C 180,E1 28806.882,E2 28806.882} C_VEL
LIN {X 0,Y 247.778,Z 645.315,A -85,B 0,C 180,E1 28817.036,E2 28817.036} C_VEL
LIN {X 0,Y 248.923,Z 689.63,A -85,B 0,C 180,E1 28838.914,E2 28838.914} C_VEL
LIN {X 0,Y 277.698,Z 720.178,A -85,B 0,C 180,E1 28857.695,E2 28857.695} C_VEL
LIN {X 0,Y 300.215,Z 738.698,A -85,B 0,C 180,E1 28868.976,E2 28868.976} C_VEL
LIN {X 0,Y 313.321,Z 750.426,A -85,B 0,C 180,E1 28877.42,E2 28877.42} C_VEL
LIN {X 0,Y 320.335,Z 756.823,A -85,B 0,C 180,E1 28885.928,E2 28885.928} C_VEL
LIN {X 0,Y 320.304,Z 756.811,A -85,B 0,C 180,E1 28894.073,E2 28894.073} C_VEL
LIN {X 0,Y 313.369,Z 750.429,A -85,B 0,C 180,E1 28902.578,E2 28902.578} C_VEL
LIN {X 0,Y 311.694,Z 748.911,A -85,B 0,C 180,E1 28903.858,E2 28903.858} C_VEL
LIN {X 0,Y 294.334,Z 742.105,A -85,B 0,C 180,E1 28909.623,E2 28909.623} C_VEL
LIN {X 0,Y 272.753,Z 725.381,A -85,B 0,C 180,E1 28920.623,E2 28920.623} C_VEL
LIN {X 0,Y 243.592,Z 697.059,A -85,B 0,C 180,E1 28939.298,E2 28939.298} C_VEL
LIN {X 0,Y 240.8,Z 658.684,A -85,B 0,C 180,E1 28959.839,E2 28959.839} C_VEL
LIN {X 0,Y 244.429,Z 640.408,A -85,B 0,C 180,E1 28970.28,E2 28970.28} C_VEL
LIN {X 0,Y 246.034,Z 634.033,A -85,B 0,C 180,E1 28978.339,E2 28978.339} C_VEL
LIN {X 0,Y 245.32,Z 638.469,A -85,B 0,C 180,E1 28987.212,E2 28987.212} C_VEL
LIN {X 0,Y 243.506,Z 654.476,A -85,B 0,C 180,E1 28997.554,E2 28997.554} C_VEL
LIN {X 0,Y 240.153,Z 665.298,A -85,B 0,C 180,E1 29001.484,E2 29001.484} C_VEL
LIN {X 0,Y 200.573,Z 710.523,A -85,B 0,C 180,E1 29009.601,E2 29009.601} C_VEL
LIN {X 0,Y 162.358,Z 743.287,A -85,B 0,C 180,E1 29023.624,E2 29023.624} C_VEL
LIN {X 0,Y 136.085,Z 763.046,A -85,B 0,C 180,E1 29047.043,E2 29047.043} C_VEL
LIN {X 0,Y 131.261,Z 767.79,A -85,B 0,C 180,E1 29066.688,E2 29066.688} C_VEL
LIN {X 0,Y 134.53,Z 764.288,A -85,B 0,C 180,E1 29089.765,E2 29089.765} C_VEL
LIN {X 0,Y 157.841,Z 746.513,A -85,B 0,C 180,E1 29113.955,E2 29113.955} C_VEL
LIN {X 0,Y 196.179,Z 714.605,A -85,B 0,C 180,E1 29129.239,E2 29129.239} C_VEL
LIN {X 0,Y 236.085,Z 670.672,A -85,B 0,C 180,E1 29137.856,E2 29137.856} C_VEL
LIN {X 0,Y 242.625,Z 660.364,A -85,B 0,C 180,E1 29139.769,E2 29139.769} C_VEL
LIN {X 0,Y 245.011,Z 642.653,A -85,B 0,C 180,E1 29149.186,E2 29149.186} C_VEL
LIN {X 0,Y 245.984,Z 634.469,A -85,B 0,C 180,E1 29158.127,E2 29158.127} C_VEL
LIN {X 0,Y 245.069,Z 636.373,A -85,B 0,C 180,E1 29165.222,E2 29165.222} C_VEL
LIN {X 0,Y 242.971,Z 648.724,A -85,B 0,C 180,E1 29175.279,E2 29175.279} C_VEL
LIN {X 0,Y 242.39,Z 694.281,A -85,B 0,C 180,E1 29199.027,E2 29199.027} C_VEL
LIN {X 0,Y 271.011,Z 723.611,A -85,B 0,C 180,E1 29218.315,E2 29218.315} C_VEL
LIN {X 0,Y 292.704,Z 740.563,A -85,B 0,C 180,E1 29229.368,E2 29229.368} C_VEL
LIN {X 0,Y 306.097,Z 751.83,A -85,B 0,C 180,E1 29238.2,E2 29238.2} C_VEL
LIN {X 0,Y 312.197,Z 757.328,A -85,B 0,C 180,E1 29245.822,E2 29245.822} C_VEL
LIN {X 0,Y 313.325,Z 758.018,A -85,B 0,C 180,E1 29251.387,E2 29251.387} C_VEL
LIN {X 0,Y 307.387,Z 752.991,A -85,B 0,C 180,E1 29260.695,E2 29260.695} C_VEL
LIN {X 0,Y 294.334,Z 742.105,A -85,B 0,C 180,E1 29269.623,E2 29269.623} C_VEL
LIN {X 0,Y 274.896,Z 735.028,A -85,B 0,C 180,E1 29275.487,E2 29275.487} C_VEL
LIN {X 0,Y 247.94,Z 713.958,A -85,B 0,C 180,E1 29290.264,E2 29290.264} C_VEL
LIN {X 0,Y 232.052,Z 676.849,A -85,B 0,C 180,E1 29314.12,E2 29314.12} C_VEL
LIN {X 0,Y 238.497,Z 651.187,A -85,B 0,C 180,E1 29327.247,E2 29327.247} C_VEL
LIN {X 0,Y 241.35,Z 640.67,A -85,B 0,C 180,E1 29338.307,E2 29338.307} C_VEL
LIN {X 0,Y 240.549,Z 645.232,A -85,B 0,C 180,E1 29347.297,E2 29347.297} C_VEL
LIN {X 0,Y 238.225,Z 659.482,A -85,B 0,C 180,E1 29356.768,E2 29356.768} C_VEL
LIN {X 0,Y 235.418,Z 667.55,A -85,B 0,C 180,E1 29359.944,E2 29359.944} C_VEL
LIN {X 0,Y 193.428,Z 713.263,A -85,B 0,C 180,E1 29368.345,E2 29368.345} C_VEL
LIN {X 0,Y 152.586,Z 746.009,A -85,B 0,C 180,E1 29383.668,E2 29383.668} C_VEL
LIN {X 0,Y 126.972,Z 764.112,A -85,B 0,C 180,E1 29409.004,E2 29409.004} C_VEL
LIN {X 0,Y 123.508,Z 767.62,A -85,B 0,C 180,E1 29433.519,E2 29433.519} C_VEL
LIN {X 0,Y 133.252,Z 759.584,A -85,B 0,C 180,E1 29460.978,E2 29460.978} C_VEL
LIN {X 0,Y 165.499,Z 736.666,A -85,B 0,C 180,E1 29482.481,E2 29482.481} C_VEL
LIN {X 0,Y 207.23,Z 700.03,A -85,B 0,C 180,E1 29494.902,E2 29494.902} C_VEL
LIN {X 0,Y 237.251,Z 664.29,A -85,B 0,C 180,E1 29500.885,E2 29500.885} C_VEL
LIN {X 0,Y 240.147,Z 648.716,A -85,B 0,C 180,E1 29509.636,E2 29509.636} C_VEL
LIN {X 0,Y 241.306,Z 641.099,A -85,B 0,C 180,E1 29518.091,E2 29518.091} C_VEL
LIN {X 0,Y 240.156,Z 643.906,A -85,B 0,C 180,E1 29526.38,E2 29526.38} C_VEL
LIN {X 0,Y 237.016,Z 657.744,A -85,B 0,C 180,E1 29536.627,E2 29536.627} C_VEL
LIN {X 0,Y 235.335,Z 697.998,A -85,B 0,C 180,E1 29558.647,E2 29558.647} C_VEL
LIN {X 0,Y 263.095,Z 726.018,A -85,B 0,C 180,E1 29578.316,E2 29578.316} C_VEL
LIN {X 0,Y 285.223,Z 742.418,A -85,B 0,C 180,E1 29589.782,E2 29589.782} C_VEL
LIN {X 0,Y 297.996,Z 752.434,A -85,B 0,C 180,E1 29598.255,E2 29598.255} C_VEL
LIN {X 0,Y 304.07,Z 757.555,A -85,B 0,C 180,E1 29605.71,E2 29605.71} C_VEL
LIN {X 0,Y 305.293,Z 758.286,A -85,B 0,C 180,E1 29611.423,E2 29611.423} C_VEL
LIN {X 0,Y 299.752,Z 753.833,A -85,B 0,C 180,E1 29620.199,E2 29620.199} C_VEL
LIN {X 0,Y 286.828,Z 743.748,A -85,B 0,C 180,E1 29629.196,E2 29629.196} C_VEL
LIN {X 0,Y 274.896,Z 735.028,A -85,B 0,C 180,E1 29635.487,E2 29635.487} C_VEL
